LIN {X 0,Y 470.196,Z 271.556,A -85,B 0,C 180,E1 -7475.307,E2 -7475.307} C_VEL
LIN {X 0,Y 469.91,Z 283.904,A -85,B 0,C 180,E1 -7475.848,E2 -7475.848} C_VEL
LIN {X 0,Y 469.494,Z 295.789,A -85,B 0,C 180,E1 -7476.554,E2 -7476.554} C_VEL
LIN {X 0,Y 469.053,Z 307.196,A -85,B 0,C 180,E1 -7477.425,E2 -7477.425} C_VEL
LIN {X 0,Y 468.572,Z 317.556,A -85,B 0,C 180,E1 -7478.415,E2 -7478.415} C_VEL
LIN {X 0,Y 468.062,Z 326.78,A -85,B 0,C 180,E1 -7479.507,E2 -7479.507} C_VEL
LIN {X 0,Y 467.676,Z 335.773,A -85,B 0,C 180,E1 -7480.827,E2 -7480.827} C_VEL
LIN {X 0,Y 467.329,Z 343.109,A -85,B 0,C 180,E1 -7482.174,E2 -7482.174} C_VEL
LIN {X 0,Y 467.061,Z 348.773,A -85,B 0,C 180,E1 -7483.488,E2 -7483.488} C_VEL
LIN {X 0,Y 466.917,Z 353.288,A -85,B 0,C 180,E1 -7484.826,E2 -7484.826} C_VEL
LIN {X 0,Y 466.808,Z 355.68,A -85,B 0,C 180,E1 -7485.724,E2 -7485.724} C_VEL
LIN {X 0,Y 466.714,Z 357.623,A -85,B 0,C 180,E1 -7486.625,E2 -7486.625} C_VEL
LIN {X 0,Y 466.631,Z 359.065,A -85,B 0,C 180,E1 -7487.531,E2 -7487.531} C_VEL
LIN {X 0,Y 466.627,Z 360.079,A -85,B 0,C 180,E1 -7488.439,E2 -7488.439} C_VEL
LIN {X 0,Y 466.597,Z 360.681,A -85,B 0,C 180,E1 -7489.352,E2 -7489.352} C_VEL
LIN {X 0,Y 466.598,Z 360.615,A -85,B 0,C 180,E1 -7490.956,E2 -7490.956} C_VEL
LIN {X 0,Y 466.631,Z 359.745,A -85,B 0,C 180,E1 -7492.119,E2 -7492.119} C_VEL
LIN {X 0,Y 466.738,Z 358.096,A -85,B 0,C 180,E1 -7493.29,E2 -7493.29} C_VEL
LIN {X 0,Y 466.878,Z 354.549,A -85,B 0,C 180,E1 -7494.929,E2 -7494.929} C_VEL
LIN {X 0,Y 467.08,Z 350.108,A -85,B 0,C 180,E1 -7496.352,E2 -7496.352} C_VEL
LIN {X 0,Y 467.309,Z 344.226,A -85,B 0,C 180,E1 -7497.789,E2 -7497.789} C_VEL
LIN {X 0,Y 467.671,Z 337.664,A -85,B 0,C 180,E1 -7499.06,E2 -7499.06} C_VEL
LIN {X 0,Y 468.03,Z 330.441,A -85,B 0,C 180,E1 -7500.202,E2 -7500.202} C_VEL
LIN {X 0,Y 468.494,Z 321.406,A -85,B 0,C 180,E1 -7501.37,E2 -7501.37} C_VEL
LIN {X 0,Y 468.951,Z 311.594,A -85,B 0,C 180,E1 -7502.397,E2 -7502.397} C_VEL
LIN {X 0,Y 469.534,Z 300.538,A -85,B 0,C 180,E1 -7503.325,E2 -7503.325} C_VEL
LIN {X 0,Y 470.053,Z 288.74,A -85,B 0,C 180,E1 -7504.103,E2 -7504.103} C_VEL
LIN {X 0,Y 470.403,Z 275.786,A -85,B 0,C 180,E1 -7504.743,E2 -7504.743} C_VEL
LIN {X 0,Y 470.731,Z 262.741,A -85,B 0,C 180,E1 -7505.191,E2 -7505.191} C_VEL
LIN {X 0,Y 470.898,Z 248.767,A -85,B 0,C 180,E1 -7505.474,E2 -7505.474} C_VEL
LIN {X 0,Y 471.517,Z 164.162,A -85,B 0,C 180,E1 -7506.79,E2 -7506.79} C_VEL
LIN {X 0,Y 468.69,Z 150.58,A -85,B 0,C 180,E1 -7507.134,E2 -7507.134} C_VEL
LIN {X 0,Y 468.755,Z 141.458,A -85,B 0,C 180,E1 -7509.028,E2 -7509.028} C_VEL
LIN {X 0,Y 467.591,Z 135.242,A -85,B 0,C 180,E1 -7510.405,E2 -7510.405} C_VEL
LIN {X 0,Y 467.544,Z 135.249,A -85,B 0,C 180,E1 -7513.82,E2 -7513.82} C_VEL
LIN {X 0,Y 467.544,Z 135.248,A -85,B 0,C 180,E1 -7516.254,E2 -7516.254} C_VEL
LIN {X 0,Y 467.557,Z 135.241,A -85,B 0,C 180,E1 -7519.733,E2 -7519.733} C_VEL
LIN {X 0,Y 467.542,Z 135.246,A -85,B 0,C 180,E1 -7522.815,E2 -7522.815} C_VEL
LIN {X 0,Y 467.576,Z 135.239,A -85,B 0,C 180,E1 -7525.76,E2 -7525.76} C_VEL
LIN {X 0,Y 467.537,Z 135.249,A -85,B 0,C 180,E1 -7528.962,E2 -7528.962} C_VEL
LIN {X 0,Y 467.543,Z 135.245,A -85,B 0,C 180,E1 -7532.226,E2 -7532.226} C_VEL
LIN {X 0,Y 467.552,Z 135.245,A -85,B 0,C 180,E1 -7535.11,E2 -7535.11} C_VEL
LIN {X 0,Y 467.518,Z 135.243,A -85,B 0,C 180,E1 -7537.926,E2 -7537.926} C_VEL
LIN {X 0,Y 467.568,Z 135.237,A -85,B 0,C 180,E1 -7541.254,E2 -7541.254} C_VEL
LIN {X 0,Y 467.577,Z 135.242,A -85,B 0,C 180,E1 -7544.303,E2 -7544.303} C_VEL
LIN {X 0,Y 467.642,Z 135.233,A -85,B 0,C 180,E1 -7547.854,E2 -7547.854} C_VEL
LIN {X 0,Y 467.63,Z 135.231,A -85,B 0,C 180,E1 -7551.356,E2 -7551.356} C_VEL
LIN {X 0,Y 467.7,Z 135.223,A -85,B 0,C 180,E1 -7553.962,E2 -7553.962} C_VEL
LIN {X 0,Y 467.811,Z 135.208,A -85,B 0,C 180,E1 -7557.417,E2 -7557.417} C_VEL
LIN {X 0,Y 467.85,Z 135.209,A -85,B 0,C 180,E1 -7560,E2 -7560} C_VEL
LIN {X 0,Y 467.813,Z 135.203,A -85,B 0,C 180,E1 -7562.583,E2 -7562.583} C_VEL
LIN {X 0,Y 467.702,Z 135.224,A -85,B 0,C 180,E1 -7566.038,E2 -7566.038} C_VEL
LIN {X 0,Y 467.637,Z 135.227,A -85,B 0,C 180,E1 -7568.644,E2 -7568.644} C_VEL
LIN {X 0,Y 467.658,Z 135.224,A -85,B 0,C 180,E1 -7572.146,E2 -7572.146} C_VEL
LIN {X 0,Y 467.639,Z 135.233,A -85,B 0,C 180,E1 -7575.695,E2 -7575.695} C_VEL
LIN {X 0,Y 467.622,Z 135.237,A -85,B 0,C 180,E1 -7579.308,E2 -7579.308} C_VEL
LIN {X 0,Y 467.536,Z 135.237,A -85,B 0,C 180,E1 -7582.074,E2 -7582.074} C_VEL
LIN {X 0,Y 467.571,Z 135.243,A -85,B 0,C 180,E1 -7584.889,E2 -7584.889} C_VEL
LIN {X 0,Y 467.564,Z 135.24,A -85,B 0,C 180,E1 -7587.773,E2 -7587.773} C_VEL
LIN {X 0,Y 467.567,Z 135.243,A -85,B 0,C 180,E1 -7591.044,E2 -7591.044} C_VEL
LIN {X 0,Y 467.579,Z 135.237,A -85,B 0,C 180,E1 -7594.24,E2 -7594.24} C_VEL
LIN {X 0,Y 467.549,Z 135.242,A -85,B 0,C 180,E1 -7597.186,E2 -7597.186} C_VEL
LIN {X 0,Y 467.561,Z 135.244,A -85,B 0,C 180,E1 -7600.267,E2 -7600.267} C_VEL
LIN {X 0,Y 467.562,Z 135.246,A -85,B 0,C 180,E1 -7602.563,E2 -7602.563} C_VEL
LIN {X 0,Y 467.568,Z 135.242,A -85,B 0,C 180,E1 -7605.052,E2 -7605.052} C_VEL
LIN {X 0,Y 467.575,Z 135.245,A -85,B 0,C 180,E1 -7608.597,E2 -7608.597} C_VEL
LIN {X 0,Y 467.565,Z 135.244,A -85,B 0,C 180,E1 -7611.955,E2 -7611.955} C_VEL
LIN {X 0,Y 467.565,Z 135.238,A -85,B 0,C 180,E1 -7615.167,E2 -7615.167} C_VEL
LIN {X 0,Y 467.585,Z 135.243,A -85,B 0,C 180,E1 -7618.26,E2 -7618.26} C_VEL
LIN {X 0,Y 467.577,Z 135.242,A -85,B 0,C 180,E1 -7621.25,E2 -7621.25} C_VEL
LIN {X 0,Y 467.658,Z 135.282,A -85,B 0,C 180,E1 -7623.443,E2 -7623.443} C_VEL
LIN {X 0,Y 470.052,Z 147.842,A -85,B 0,C 180,E1 -7625.79,E2 -7625.79} C_VEL
LIN {X 0,Y 469.273,Z 165.112,A -85,B 0,C 180,E1 -7628.74,E2 -7628.74} C_VEL
LIN {X 0,Y 468.539,Z 183.705,A -85,B 0,C 180,E1 -7631.865,E2 -7631.865} C_VEL
LIN {X 0,Y 468.302,Z 189.868,A -85,B 0,C 180,E1 -7632.89,E2 -7632.89} C_VEL
LIN {X 0,Y 471.264,Z 209.86,A -85,B 0,C 180,E1 -7633.329,E2 -7633.329} C_VEL
LIN {X 0,Y 470.584,Z 299.18,A -85,B 0,C 180,E1 -7634.738,E2 -7634.738} C_VEL
LIN {X 0,Y 470.197,Z 312.223,A -85,B 0,C 180,E1 -7635.114,E2 -7635.114} C_VEL
LIN {X 0,Y 469.718,Z 324.844,A -85,B 0,C 180,E1 -7635.652,E2 -7635.652} C_VEL
LIN {X 0,Y 469.153,Z 336.885,A -85,B 0,C 180,E1 -7636.353,E2 -7636.353} C_VEL
LIN {X 0,Y 468.684,Z 347.532,A -85,B 0,C 180,E1 -7637.148,E2 -7637.148} C_VEL
LIN {X 0,Y 468.152,Z 358.788,A -85,B 0,C 180,E1 -7638.197,E2 -7638.197} C_VEL
LIN {X 0,Y 467.73,Z 367.295,A -85,B 0,C 180,E1 -7639.174,E2 -7639.174} C_VEL
LIN {X 0,Y 467.361,Z 375.155,A -85,B 0,C 180,E1 -7640.26,E2 -7640.26} C_VEL
LIN {X 0,Y 467.081,Z 382.844,A -85,B 0,C 180,E1 -7641.564,E2 -7641.564} C_VEL
LIN {X 0,Y 466.829,Z 389.953,A -85,B 0,C 180,E1 -7643.082,E2 -7643.082} C_VEL
LIN {X 0,Y 466.726,Z 394.684,A -85,B 0,C 180,E1 -7644.383,E2 -7644.383} C_VEL
LIN {X 0,Y 466.647,Z 398.301,A -85,B 0,C 180,E1 -7645.681,E2 -7645.681} C_VEL
LIN {X 0,Y 466.7,Z 400.168,A -85,B 0,C 180,E1 -7646.547,E2 -7646.547} C_VEL
LIN {X 0,Y 466.685,Z 401.568,A -85,B 0,C 180,E1 -7647.41,E2 -7647.41} C_VEL
LIN {X 0,Y 466.662,Z 402.568,A -85,B 0,C 180,E1 -7648.274,E2 -7648.274} C_VEL
LIN {X 0,Y 466.627,Z 403.178,A -85,B 0,C 180,E1 -7649.137,E2 -7649.137} C_VEL
LIN {X 0,Y 466.611,Z 403.388,A -85,B 0,C 180,E1 -7650,E2 -7650} C_VEL
LIN {X 0,Y 466.662,Z 402.552,A -85,B 0,C 180,E1 -7651.726,E2 -7651.726} C_VEL
LIN {X 0,Y 466.685,Z 401.548,A -85,B 0,C 180,E1 -7652.589,E2 -7652.589} C_VEL
LIN {X 0,Y 466.7,Z 400.131,A -85,B 0,C 180,E1 -7653.453,E2 -7653.453} C_VEL
LIN {X 0,Y 466.687,Z 397.162,A -85,B 0,C 180,E1 -7654.751,E2 -7654.751} C_VEL
LIN {X 0,Y 466.712,Z 392.03,A -85,B 0,C 180,E1 -7656.349,E2 -7656.349} C_VEL
LIN {X 0,Y 466.931,Z 385.925,A -85,B 0,C 180,E1 -7657.785,E2 -7657.785} C_VEL
LIN {X 0,Y 467.169,Z 378.933,A -85,B 0,C 180,E1 -7659.088,E2 -7659.088} C_VEL
LIN {X 0,Y 467.522,Z 370.162,A -85,B 0,C 180,E1 -7660.392,E2 -7660.392} C_VEL
LIN {X 0,Y 467.984,Z 361.182,A -85,B 0,C 180,E1 -7661.477,E2 -7661.477} C_VEL
LIN {X 0,Y 468.438,Z 350.306,A -85,B 0,C 180,E1 -7662.546,E2 -7662.546} C_VEL
LIN {X 0,Y 468.963,Z 338.844,A -85,B 0,C 180,E1 -7663.432,E2 -7663.432} C_VEL
LIN {X 0,Y 469.526,Z 326.234,A -85,B 0,C 180,E1 -7664.188,E2 -7664.188} C_VEL
LIN {X 0,Y 469.867,Z 315.464,A -85,B 0,C 180,E1 -7664.675,E2 -7664.675} C_VEL
LIN {X 0,Y 470.257,Z 302.801,A -85,B 0,C 180,E1 -7665.078,E2 -7665.078} C_VEL
LIN {X 0,Y 470.533,Z 286.718,A -85,B 0,C 180,E1 -7665.374,E2 -7665.374} C_VEL
LIN {X 0,Y 470.903,Z 208.82,A -85,B 0,C 180,E1 -7666.579,E2 -7666.579} C_VEL
LIN {X 0,Y 468.236,Z 190.139,A -85,B 0,C 180,E1 -7666.987,E2 -7666.987} C_VEL
LIN {X 0,Y 468.855,Z 172.415,A -85,B 0,C 180,E1 -7669.939,E2 -7669.939} C_VEL
LIN {X 0,Y 469.666,Z 153.43,A -85,B 0,C 180,E1 -7673.129,E2 -7673.129} C_VEL
LIN {X 0,Y 469.904,Z 147.289,A -85,B 0,C 180,E1 -7674.17,E2 -7674.17} C_VEL
LIN {X 0,Y 467.654,Z 135.235,A -85,B 0,C 180,E1 -7676.377,E2 -7676.377} C_VEL
LIN {X 0,Y 467.57,Z 135.242,A -85,B 0,C 180,E1 -7679.332,E2 -7679.332} C_VEL
LIN {X 0,Y 467.583,Z 135.237,A -85,B 0,C 180,E1 -7682.679,E2 -7682.679} C_VEL
LIN {X 0,Y 467.561,Z 135.245,A -85,B 0,C 180,E1 -7685.739,E2 -7685.739} C_VEL
LIN {X 0,Y 467.583,Z 135.237,A -85,B 0,C 180,E1 -7689.144,E2 -7689.144} C_VEL
LIN {X 0,Y 467.588,Z 135.236,A -85,B 0,C 180,E1 -7692.567,E2 -7692.567} C_VEL
LIN {X 0,Y 467.567,Z 135.239,A -85,B 0,C 180,E1 -7695.052,E2 -7695.052} C_VEL
LIN {X 0,Y 467.59,Z 135.241,A -85,B 0,C 180,E1 -7697.44,E2 -7697.44} C_VEL
LIN {X 0,Y 467.561,Z 135.24,A -85,B 0,C 180,E1 -7700.853,E2 -7700.853} C_VEL
LIN {X 0,Y 467.559,Z 135.24,A -85,B 0,C 180,E1 -7704.261,E2 -7704.261} C_VEL
LIN {X 0,Y 467.58,Z 135.243,A -85,B 0,C 180,E1 -7707.321,E2 -7707.321} C_VEL
LIN {X 0,Y 467.569,Z 135.239,A -85,B 0,C 180,E1 -7710.667,E2 -7710.667} C_VEL
LIN {X 0,Y 467.616,Z 135.239,A -85,B 0,C 180,E1 -7713.199,E2 -7713.199} C_VEL
LIN {X 0,Y 467.593,Z 135.236,A -85,B 0,C 180,E1 -7716.468,E2 -7716.468} C_VEL
LIN {X 0,Y 467.623,Z 135.232,A -85,B 0,C 180,E1 -7719.777,E2 -7719.777} C_VEL
LIN {X 0,Y 467.598,Z 135.236,A -85,B 0,C 180,E1 -7722.506,E2 -7722.506} C_VEL
LIN {X 0,Y 467.607,Z 135.239,A -85,B 0,C 180,E1 -7725.196,E2 -7725.196} C_VEL
LIN {X 0,Y 467.656,Z 135.227,A -85,B 0,C 180,E1 -7727.854,E2 -7727.854} C_VEL
LIN {X 0,Y 467.669,Z 135.228,A -85,B 0,C 180,E1 -7731.357,E2 -7731.357} C_VEL
LIN {X 0,Y 467.724,Z 135.219,A -85,B 0,C 180,E1 -7733.962,E2 -7733.962} C_VEL
LIN {X 0,Y 467.859,Z 135.203,A -85,B 0,C 180,E1 -7737.417,E2 -7737.417} C_VEL
LIN {X 0,Y 467.882,Z 135.2,A -85,B 0,C 180,E1 -7740,E2 -7740} C_VEL
LIN {X 0,Y 467.859,Z 135.21,A -85,B 0,C 180,E1 -7742.583,E2 -7742.583} C_VEL
LIN {X 0,Y 467.735,Z 135.219,A -85,B 0,C 180,E1 -7746.037,E2 -7746.037} C_VEL
LIN {X 0,Y 467.68,Z 135.23,A -85,B 0,C 180,E1 -7748.643,E2 -7748.643} C_VEL
LIN {X 0,Y 467.656,Z 135.232,A -85,B 0,C 180,E1 -7752.145,E2 -7752.145} C_VEL
LIN {X 0,Y 467.638,Z 135.23,A -85,B 0,C 180,E1 -7755.695,E2 -7755.695} C_VEL
LIN {X 0,Y 467.621,Z 135.231,A -85,B 0,C 180,E1 -7759.308,E2 -7759.308} C_VEL
LIN {X 0,Y 467.534,Z 135.249,A -85,B 0,C 180,E1 -7762.074,E2 -7762.074} C_VEL
LIN {X 0,Y 467.585,Z 135.236,A -85,B 0,C 180,E1 -7764.888,E2 -7764.888} C_VEL
LIN {X 0,Y 467.618,Z 135.236,A -85,B 0,C 180,E1 -7767.769,E2 -7767.769} C_VEL
LIN {X 0,Y 467.567,Z 135.238,A -85,B 0,C 180,E1 -7771.045,E2 -7771.045} C_VEL
LIN {X 0,Y 467.587,Z 135.239,A -85,B 0,C 180,E1 -7774.242,E2 -7774.242} C_VEL
LIN {X 0,Y 467.547,Z 135.242,A -85,B 0,C 180,E1 -7777.186,E2 -7777.186} C_VEL
LIN {X 0,Y 467.576,Z 135.239,A -85,B 0,C 180,E1 -7780.265,E2 -7780.265} C_VEL
LIN {X 0,Y 467.585,Z 135.236,A -85,B 0,C 180,E1 -7782.567,E2 -7782.567} C_VEL
LIN {X 0,Y 467.565,Z 135.24,A -85,B 0,C 180,E1 -7785.053,E2 -7785.053} C_VEL
LIN {X 0,Y 467.588,Z 135.242,A -85,B 0,C 180,E1 -7787.44,E2 -7787.44} C_VEL
LIN {X 0,Y 467.559,Z 135.24,A -85,B 0,C 180,E1 -7790.853,E2 -7790.853} C_VEL
LIN {X 0,Y 467.558,Z 135.24,A -85,B 0,C 180,E1 -7794.261,E2 -7794.261} C_VEL
LIN {X 0,Y 467.578,Z 135.244,A -85,B 0,C 180,E1 -7797.322,E2 -7797.322} C_VEL
LIN {X 0,Y 467.568,Z 135.239,A -85,B 0,C 180,E1 -7800.668,E2 -7800.668} C_VEL
LIN {X 0,Y 467.615,Z 135.24,A -85,B 0,C 180,E1 -7803.2,E2 -7803.2} C_VEL
LIN {X 0,Y 467.592,Z 135.236,A -85,B 0,C 180,E1 -7806.468,E2 -7806.468} C_VEL
LIN {X 0,Y 467.622,Z 135.232,A -85,B 0,C 180,E1 -7809.777,E2 -7809.777} C_VEL
LIN {X 0,Y 467.598,Z 135.236,A -85,B 0,C 180,E1 -7812.507,E2 -7812.507} C_VEL
LIN {X 0,Y 467.605,Z 135.239,A -85,B 0,C 180,E1 -7815.197,E2 -7815.197} C_VEL
LIN {X 0,Y 467.596,Z 135.237,A -85,B 0,C 180,E1 -7815.422,E2 -7815.422} C_VEL
LIN {X 0,Y 466.925,Z 135.319,A -85,B 0,C 180,E1 -7816.141,E2 -7816.141} C_VEL
LIN {X 0,Y 464.082,Z 135.676,A -85,B 0,C 180,E1 -7817.309,E2 -7817.309} C_VEL
LIN {X 0,Y 461.683,Z 135.973,A -85,B 0,C 180,E1 -7818.252,E2 -7818.252} C_VEL
LIN {X 0,Y 460.656,Z 136.106,A -85,B 0,C 180,E1 -7818.979,E2 -7818.979} C_VEL
LIN {X 0,Y 460.574,Z 136.11,A -85,B 0,C 180,E1 -7819.226,E2 -7819.226} C_VEL
LIN {X 0,Y 460.669,Z 136.103,A -85,B 0,C 180,E1 -7822.587,E2 -7822.587} C_VEL
LIN {X 0,Y 460.691,Z 136.103,A -85,B 0,C 180,E1 -7824.748,E2 -7824.748} C_VEL
LIN {X 0,Y 460.8,Z 136.086,A -85,B 0,C 180,E1 -7827.378,E2 -7827.378} C_VEL
LIN {X 0,Y 460.832,Z 136.088,A -85,B 0,C 180,E1 -7829.782,E2 -7829.782} C_VEL
LIN {X 0,Y 461.668,Z 143.128,A -85,B 0,C 180,E1 -7831.309,E2 -7831.309} C_VEL
LIN {X 0,Y 461.465,Z 150.576,A -85,B 0,C 180,E1 -7832.865,E2 -7832.865} C_VEL
LIN {X 0,Y 464.479,Z 166.22,A -85,B 0,C 180,E1 -7833.232,E2 -7833.232} C_VEL
LIN {X 0,Y 463.61,Z 257.402,A -85,B 0,C 180,E1 -7834.674,E2 -7834.674} C_VEL
LIN {X 0,Y 463.342,Z 270.667,A -85,B 0,C 180,E1 -7835.058,E2 -7835.058} C_VEL
LIN {X 0,Y 463.017,Z 283.365,A -85,B 0,C 180,E1 -7835.608,E2 -7835.608} C_VEL
LIN {X 0,Y 462.596,Z 295.48,A -85,B 0,C 180,E1 -7836.324,E2 -7836.324} C_VEL
LIN {X 0,Y 462.151,Z 306.991,A -85,B 0,C 180,E1 -7837.207,E2 -7837.207} C_VEL
LIN {X 0,Y 461.621,Z 316.821,A -85,B 0,C 180,E1 -7838.144,E2 -7838.144} C_VEL
LIN {X 0,Y 461.147,Z 325.936,A -85,B 0,C 180,E1 -7839.208,E2 -7839.208} C_VEL
LIN {X 0,Y 460.665,Z 335.146,A -85,B 0,C 180,E1 -7840.549,E2 -7840.549} C_VEL
LIN {X 0,Y 460.321,Z 342.28,A -85,B 0,C 180,E1 -7841.839,E2 -7841.839} C_VEL
LIN {X 0,Y 460.047,Z 348.506,A -85,B 0,C 180,E1 -7843.247,E2 -7843.247} C_VEL
LIN {X 0,Y 459.876,Z 353.163,A -85,B 0,C 180,E1 -7844.605,E2 -7844.605} C_VEL
LIN {X 0,Y 459.702,Z 356.698,A -85,B 0,C 180,E1 -7845.973,E2 -7845.973} C_VEL
LIN {X 0,Y 459.603,Z 358.447,A -85,B 0,C 180,E1 -7846.89,E2 -7846.89} C_VEL
LIN {X 0,Y 459.543,Z 360.487,A -85,B 0,C 180,E1 -7848.524,E2 -7848.524} C_VEL
LIN {X 0,Y 459.514,Z 361.075,A -85,B 0,C 180,E1 -7849.663,E2 -7849.663} C_VEL
LIN {X 0,Y 459.508,Z 360.881,A -85,B 0,C 180,E1 -7851.098,E2 -7851.098} C_VEL
LIN {X 0,Y 459.558,Z 359.697,A -85,B 0,C 180,E1 -7852.478,E2 -7852.478} C_VEL
LIN {X 0,Y 459.671,Z 358.257,A -85,B 0,C 180,E1 -7853.458,E2 -7853.458} C_VEL
LIN {X 0,Y 459.815,Z 355.292,A -85,B 0,C 180,E1 -7854.855,E2 -7854.855} C_VEL
LIN {X 0,Y 459.998,Z 351.028,A -85,B 0,C 180,E1 -7856.3,E2 -7856.3} C_VEL
LIN {X 0,Y 460.273,Z 344.609,A -85,B 0,C 180,E1 -7857.913,E2 -7857.913} C_VEL
LIN {X 0,Y 460.675,Z 337.949,A -85,B 0,C 180,E1 -7859.222,E2 -7859.222} C_VEL
LIN {X 0,Y 461.098,Z 330.249,A -85,B 0,C 180,E1 -7860.451,E2 -7860.451} C_VEL
LIN {X 0,Y 461.571,Z 321.633,A -85,B 0,C 180,E1 -7861.57,E2 -7861.57} C_VEL
LIN {X 0,Y 462.068,Z 311.08,A -85,B 0,C 180,E1 -7862.68,E2 -7862.68} C_VEL
LIN {X 0,Y 462.68,Z 300.588,A -85,B 0,C 180,E1 -7863.563,E2 -7863.563} C_VEL
LIN {X 0,Y 463.214,Z 288.767,A -85,B 0,C 180,E1 -7864.348,E2 -7864.348} C_VEL
LIN {X 0,Y 463.58,Z 275.971,A -85,B 0,C 180,E1 -7864.986,E2 -7864.986} C_VEL
LIN {X 0,Y 463.925,Z 262.705,A -85,B 0,C 180,E1 -7865.445,E2 -7865.445} C_VEL
LIN {X 0,Y 464.126,Z 247.598,A -85,B 0,C 180,E1 -7865.744,E2 -7865.744} C_VEL
LIN {X 0,Y 464.845,Z 165.396,A -85,B 0,C 180,E1 -7867.043,E2 -7867.043} C_VEL
LIN {X 0,Y 461.776,Z 150.914,A -85,B 0,C 180,E1 -7867.423,E2 -7867.423} C_VEL
LIN {X 0,Y 461.848,Z 142.925,A -85,B 0,C 180,E1 -7869.098,E2 -7869.098} C_VEL
LIN {X 0,Y 460.523,Z 136.122,A -85,B 0,C 180,E1 -7870.62,E2 -7870.62} C_VEL
LIN {X 0,Y 460.504,Z 136.124,A -85,B 0,C 180,E1 -7874.169,E2 -7874.169} C_VEL
LIN {X 0,Y 460.462,Z 136.131,A -85,B 0,C 180,E1 -7877.107,E2 -7877.107} C_VEL
LIN {X 0,Y 460.513,Z 136.117,A -85,B 0,C 180,E1 -7880.136,E2 -7880.136} C_VEL
LIN {X 0,Y 460.472,Z 136.122,A -85,B 0,C 180,E1 -7883.47,E2 -7883.47} C_VEL
LIN {X 0,Y 460.516,Z 136.122,A -85,B 0,C 180,E1 -7886.674,E2 -7886.674} C_VEL
LIN {X 0,Y 460.493,Z 136.123,A -85,B 0,C 180,E1 -7889.759,E2 -7889.759} C_VEL
LIN {X 0,Y 460.489,Z 136.13,A -85,B 0,C 180,E1 -7892.751,E2 -7892.751} C_VEL
LIN {X 0,Y 460.512,Z 136.12,A -85,B 0,C 180,E1 -7895.666,E2 -7895.666} C_VEL
LIN {X 0,Y 460.51,Z 136.124,A -85,B 0,C 180,E1 -7898.583,E2 -7898.583} C_VEL
LIN {X 0,Y 460.526,Z 136.114,A -85,B 0,C 180,E1 -7901.308,E2 -7901.308} C_VEL
LIN {X 0,Y 460.521,Z 136.121,A -85,B 0,C 180,E1 -7904.056,E2 -7904.056} C_VEL
LIN {X 0,Y 460.602,Z 136.108,A -85,B 0,C 180,E1 -7907.666,E2 -7907.666} C_VEL
LIN {X 0,Y 460.585,Z 136.109,A -85,B 0,C 180,E1 -7911.223,E2 -7911.223} C_VEL
LIN {X 0,Y 460.667,Z 136.098,A -85,B 0,C 180,E1 -7913.87,E2 -7913.87} C_VEL
LIN {X 0,Y 460.755,Z 136.087,A -85,B 0,C 180,E1 -7917.377,E2 -7917.377} C_VEL
LIN {X 0,Y 460.819,Z 136.085,A -85,B 0,C 180,E1 -7920,E2 -7920} C_VEL
LIN {X 0,Y 460.756,Z 136.081,A -85,B 0,C 180,E1 -7922.623,E2 -7922.623} C_VEL
LIN {X 0,Y 460.668,Z 136.099,A -85,B 0,C 180,E1 -7926.131,E2 -7926.131} C_VEL
LIN {X 0,Y 460.595,Z 136.104,A -85,B 0,C 180,E1 -7928.777,E2 -7928.777} C_VEL
LIN {X 0,Y 460.612,Z 136.101,A -85,B 0,C 180,E1 -7932.334,E2 -7932.334} C_VEL
LIN {X 0,Y 460.581,Z 136.109,A -85,B 0,C 180,E1 -7935.988,E2 -7935.988} C_VEL
LIN {X 0,Y 460.568,Z 136.114,A -85,B 0,C 180,E1 -7939.616,E2 -7939.616} C_VEL
LIN {X 0,Y 460.512,Z 136.113,A -85,B 0,C 180,E1 -7942.429,E2 -7942.429} C_VEL
LIN {X 0,Y 460.549,Z 136.111,A -85,B 0,C 180,E1 -7945.797,E2 -7945.797} C_VEL
LIN {X 0,Y 460.517,Z 136.117,A -85,B 0,C 180,E1 -7948.236,E2 -7948.236} C_VEL
LIN {X 0,Y 460.522,Z 136.12,A -85,B 0,C 180,E1 -7951.283,E2 -7951.283} C_VEL
LIN {X 0,Y 460.525,Z 136.118,A -85,B 0,C 180,E1 -7954.504,E2 -7954.504} C_VEL
LIN {X 0,Y 460.503,Z 136.118,A -85,B 0,C 180,E1 -7957.623,E2 -7957.623} C_VEL
LIN {X 0,Y 460.527,Z 136.12,A -85,B 0,C 180,E1 -7960.267,E2 -7960.267} C_VEL
LIN {X 0,Y 460.51,Z 136.119,A -85,B 0,C 180,E1 -7963.374,E2 -7963.374} C_VEL
LIN {X 0,Y 460.511,Z 136.126,A -85,B 0,C 180,E1 -7966.626,E2 -7966.626} C_VEL
LIN {X 0,Y 460.537,Z 136.119,A -85,B 0,C 180,E1 -7969.732,E2 -7969.732} C_VEL
LIN {X 0,Y 460.499,Z 136.121,A -85,B 0,C 180,E1 -7972.524,E2 -7972.524} C_VEL
LIN {X 0,Y 460.548,Z 136.114,A -85,B 0,C 180,E1 -7975.624,E2 -7975.624} C_VEL
LIN {X 0,Y 460.54,Z 136.119,A -85,B 0,C 180,E1 -7978.745,E2 -7978.745} C_VEL
LIN {X 0,Y 460.583,Z 136.115,A -85,B 0,C 180,E1 -7982.254,E2 -7982.254} C_VEL
LIN {X 0,Y 460.59,Z 136.157,A -85,B 0,C 180,E1 -7983.187,E2 -7983.187} C_VEL
LIN {X 0,Y 463.079,Z 148.727,A -85,B 0,C 180,E1 -7985.589,E2 -7985.589} C_VEL
LIN {X 0,Y 462.484,Z 162.398,A -85,B 0,C 180,E1 -7987.968,E2 -7987.968} C_VEL
LIN {X 0,Y 461.635,Z 182.163,A -85,B 0,C 180,E1 -7991.355,E2 -7991.355} C_VEL
LIN {X 0,Y 461.33,Z 189.52,A -85,B 0,C 180,E1 -7992.603,E2 -7992.603} C_VEL
LIN {X 0,Y 464.487,Z 210.587,A -85,B 0,C 180,E1 -7993.078,E2 -7993.078} C_VEL
LIN {X 0,Y 463.803,Z 298.364,A -85,B 0,C 180,E1 -7994.482,E2 -7994.482} C_VEL
LIN {X 0,Y 463.352,Z 311.564,A -85,B 0,C 180,E1 -7994.86,E2 -7994.86} C_VEL
LIN {X 0,Y 462.836,Z 324.826,A -85,B 0,C 180,E1 -7995.434,E2 -7995.434} C_VEL
LIN {X 0,Y 462.238,Z 336.776,A -85,B 0,C 180,E1 -7996.145,E2 -7996.145} C_VEL
LIN {X 0,Y 461.758,Z 347.116,A -85,B 0,C 180,E1 -7996.929,E2 -7996.929} C_VEL
LIN {X 0,Y 461.225,Z 357.534,A -85,B 0,C 180,E1 -7997.906,E2 -7997.906} C_VEL
LIN {X 0,Y 460.743,Z 367.089,A -85,B 0,C 180,E1 -7999.008,E2 -7999.008} C_VEL
LIN {X 0,Y 460.262,Z 376.295,A -85,B 0,C 180,E1 -8000.33,E2 -8000.33} C_VEL
LIN {X 0,Y 459.964,Z 383.721,A -85,B 0,C 180,E1 -8001.654,E2 -8001.654} C_VEL
LIN {X 0,Y 459.741,Z 389.689,A -85,B 0,C 180,E1 -8002.975,E2 -8002.975} C_VEL
LIN {X 0,Y 459.625,Z 394.408,A -85,B 0,C 180,E1 -8004.296,E2 -8004.296} C_VEL
LIN {X 0,Y 459.565,Z 398.013,A -85,B 0,C 180,E1 -8005.615,E2 -8005.615} C_VEL
LIN {X 0,Y 459.596,Z 399.87,A -85,B 0,C 180,E1 -8006.493,E2 -8006.493} C_VEL
LIN {X 0,Y 459.605,Z 401.263,A -85,B 0,C 180,E1 -8007.371,E2 -8007.371} C_VEL
LIN {X 0,Y 459.56,Z 402.863,A -85,B 0,C 180,E1 -8009.124,E2 -8009.124} C_VEL
LIN {X 0,Y 459.542,Z 403.063,A -85,B 0,C 180,E1 -8010,E2 -8010} C_VEL
LIN {X 0,Y 459.56,Z 402.833,A -85,B 0,C 180,E1 -8010.876,E2 -8010.876} C_VEL
LIN {X 0,Y 459.605,Z 401.204,A -85,B 0,C 180,E1 -8012.629,E2 -8012.629} C_VEL
LIN {X 0,Y 459.597,Z 399.774,A -85,B 0,C 180,E1 -8013.507,E2 -8013.507} C_VEL
LIN {X 0,Y 459.614,Z 396.793,A -85,B 0,C 180,E1 -8014.824,E2 -8014.824} C_VEL
LIN {X 0,Y 459.635,Z 392.029,A -85,B 0,C 180,E1 -8016.342,E2 -8016.342} C_VEL
LIN {X 0,Y 459.867,Z 385.519,A -85,B 0,C 180,E1 -8017.906,E2 -8017.906} C_VEL
LIN {X 0,Y 460.104,Z 378.501,A -85,B 0,C 180,E1 -8019.229,E2 -8019.229} C_VEL
LIN {X 0,Y 460.496,Z 369.702,A -85,B 0,C 180,E1 -8020.553,E2 -8020.553} C_VEL
LIN {X 0,Y 461.057,Z 359.711,A -85,B 0,C 180,E1 -8021.764,E2 -8021.764} C_VEL
LIN {X 0,Y 461.461,Z 349.611,A -85,B 0,C 180,E1 -8022.752,E2 -8022.752} C_VEL
LIN {X 0,Y 462.017,Z 338.251,A -85,B 0,C 180,E1 -8023.637,E2 -8023.637} C_VEL
LIN {X 0,Y 462.585,Z 325.566,A -85,B 0,C 180,E1 -8024.405,E2 -8024.405} C_VEL
LIN {X 0,Y 463.059,Z 313.187,A -85,B 0,C 180,E1 -8024.952,E2 -8024.952} C_VEL
LIN {X 0,Y 463.496,Z 300.581,A -85,B 0,C 180,E1 -8025.331,E2 -8025.331} C_VEL
LIN {X 0,Y 463.717,Z 279.848,A -85,B 0,C 180,E1 -8025.69,E2 -8025.69} C_VEL
LIN {X 0,Y 464.044,Z 209.571,A -85,B 0,C 180,E1 -8026.796,E2 -8026.796} C_VEL
LIN {X 0,Y 461.224,Z 189.903,A -85,B 0,C 180,E1 -8027.224,E2 -8027.224} C_VEL
LIN {X 0,Y 461.85,Z 171.964,A -85,B 0,C 180,E1 -8030.254,E2 -8030.254} C_VEL
LIN {X 0,Y 462.717,Z 154.319,A -85,B 0,C 180,E1 -8033.26,E2 -8033.26} C_VEL
LIN {X 0,Y 462.864,Z 148.003,A -85,B 0,C 180,E1 -8034.352,E2 -8034.352} C_VEL
LIN {X 0,Y 460.616,Z 136.111,A -85,B 0,C 180,E1 -8036.567,E2 -8036.567} C_VEL
LIN {X 0,Y 460.532,Z 136.12,A -85,B 0,C 180,E1 -8039.558,E2 -8039.558} C_VEL
LIN {X 0,Y 460.533,Z 136.119,A -85,B 0,C 180,E1 -8042.284,E2 -8042.284} C_VEL
LIN {X 0,Y 460.511,Z 136.119,A -85,B 0,C 180,E1 -8045.445,E2 -8045.445} C_VEL
LIN {X 0,Y 460.546,Z 136.113,A -85,B 0,C 180,E1 -8048.897,E2 -8048.897} C_VEL
LIN {X 0,Y 460.524,Z 136.119,A -85,B 0,C 180,E1 -8052.181,E2 -8052.181} C_VEL
LIN {X 0,Y 460.515,Z 136.121,A -85,B 0,C 180,E1 -8055.411,E2 -8055.411} C_VEL
LIN {X 0,Y 460.533,Z 136.115,A -85,B 0,C 180,E1 -8058.397,E2 -8058.397} C_VEL
LIN {X 0,Y 460.519,Z 136.12,A -85,B 0,C 180,E1 -8061.266,E2 -8061.266} C_VEL
LIN {X 0,Y 460.509,Z 136.118,A -85,B 0,C 180,E1 -8064.554,E2 -8064.554} C_VEL
LIN {X 0,Y 460.53,Z 136.119,A -85,B 0,C 180,E1 -8067.715,E2 -8067.715} C_VEL
LIN {X 0,Y 460.54,Z 136.115,A -85,B 0,C 180,E1 -8070.769,E2 -8070.769} C_VEL
LIN {X 0,Y 460.56,Z 136.114,A -85,B 0,C 180,E1 -8073.734,E2 -8073.734} C_VEL
LIN {X 0,Y 460.546,Z 136.114,A -85,B 0,C 180,E1 -8076.624,E2 -8076.624} C_VEL
LIN {X 0,Y 460.552,Z 136.116,A -85,B 0,C 180,E1 -8079.453,E2 -8079.453} C_VEL
LIN {X 0,Y 460.549,Z 136.113,A -85,B 0,C 180,E1 -8082.23,E2 -8082.23} C_VEL
LIN {X 0,Y 460.566,Z 136.118,A -85,B 0,C 180,E1 -8084.965,E2 -8084.965} C_VEL
LIN {X 0,Y 460.61,Z 136.108,A -85,B 0,C 180,E1 -8088.559,E2 -8088.559} C_VEL
LIN {X 0,Y 460.619,Z 136.107,A -85,B 0,C 180,E1 -8091.224,E2 -8091.224} C_VEL
LIN {X 0,Y 460.688,Z 136.095,A -85,B 0,C 180,E1 -8093.87,E2 -8093.87} C_VEL
LIN {X 0,Y 460.8,Z 136.082,A -85,B 0,C 180,E1 -8097.377,E2 -8097.377} C_VEL
LIN {X 0,Y 460.853,Z 136.075,A -85,B 0,C 180,E1 -8100,E2 -8100} C_VEL
LIN {X 0,Y 460.824,Z 136.087,A -85,B 0,C 180,E1 -8102.622,E2 -8102.622} C_VEL
LIN {X 0,Y 460.701,Z 136.096,A -85,B 0,C 180,E1 -8106.13,E2 -8106.13} C_VEL
LIN {X 0,Y 460.627,Z 136.107,A -85,B 0,C 180,E1 -8108.776,E2 -8108.776} C_VEL
LIN {X 0,Y 460.613,Z 136.112,A -85,B 0,C 180,E1 -8112.445,E2 -8112.445} C_VEL
LIN {X 0,Y 460.6,Z 136.11,A -85,B 0,C 180,E1 -8115.997,E2 -8115.997} C_VEL
LIN {X 0,Y 460.567,Z 136.111,A -85,B 0,C 180,E1 -8119.615,E2 -8119.615} C_VEL
LIN {X 0,Y 460.51,Z 136.122,A -85,B 0,C 180,E1 -8122.429,E2 -8122.429} C_VEL
LIN {X 0,Y 460.552,Z 136.116,A -85,B 0,C 180,E1 -8125.798,E2 -8125.798} C_VEL
LIN {X 0,Y 460.55,Z 136.118,A -85,B 0,C 180,E1 -8128.233,E2 -8128.233} C_VEL
LIN {X 0,Y 460.519,Z 136.117,A -85,B 0,C 180,E1 -8131.283,E2 -8131.283} C_VEL
LIN {X 0,Y 460.53,Z 136.116,A -85,B 0,C 180,E1 -8134.505,E2 -8134.505} C_VEL
LIN {X 0,Y 460.5,Z 136.124,A -85,B 0,C 180,E1 -8137.623,E2 -8137.623} C_VEL
LIN {X 0,Y 460.541,Z 136.116,A -85,B 0,C 180,E1 -8140.269,E2 -8140.269} C_VEL
LIN {X 0,Y 460.497,Z 136.123,A -85,B 0,C 180,E1 -8143.376,E2 -8143.376} C_VEL
LIN {X 0,Y 460.497,Z 136.119,A -85,B 0,C 180,E1 -8146.625,E2 -8146.625} C_VEL
LIN {X 0,Y 460.538,Z 136.12,A -85,B 0,C 180,E1 -8149.731,E2 -8149.731} C_VEL
LIN {X 0,Y 460.498,Z 136.119,A -85,B 0,C 180,E1 -8152.524,E2 -8152.524} C_VEL
LIN {X 0,Y 460.536,Z 136.119,A -85,B 0,C 180,E1 -8155.623,E2 -8155.623} C_VEL
LIN {X 0,Y 460.536,Z 136.115,A -85,B 0,C 180,E1 -8158.745,E2 -8158.745} C_VEL
LIN {X 0,Y 460.58,Z 136.109,A -85,B 0,C 180,E1 -8162.254,E2 -8162.254} C_VEL
LIN {X 0,Y 460.546,Z 136.115,A -85,B 0,C 180,E1 -8164.705,E2 -8164.705} C_VEL
LIN {X 0,Y 460.51,Z 136.12,A -85,B 0,C 180,E1 -8167.571,E2 -8167.571} C_VEL
LIN {X 0,Y 460.568,Z 136.111,A -85,B 0,C 180,E1 -8170.385,E2 -8170.385} C_VEL
LIN {X 0,Y 460.604,Z 136.106,A -85,B 0,C 180,E1 -8174.059,E2 -8174.059} C_VEL
LIN {X 0,Y 460.609,Z 136.106,A -85,B 0,C 180,E1 -8177.666,E2 -8177.666} C_VEL
LIN {X 0,Y 460.574,Z 136.11,A -85,B 0,C 180,E1 -8179.226,E2 -8179.226} C_VEL
LIN {X 0,Y 459.911,Z 136.195,A -85,B 0,C 180,E1 -8179.955,E2 -8179.955} C_VEL
LIN {X 0,Y 457.07,Z 136.556,A -85,B 0,C 180,E1 -8181.141,E2 -8181.141} C_VEL
LIN {X 0,Y 454.679,Z 136.855,A -85,B 0,C 180,E1 -8182.098,E2 -8182.098} C_VEL
LIN {X 0,Y 453.669,Z 136.977,A -85,B 0,C 180,E1 -8182.836,E2 -8182.836} C_VEL
LIN {X 0,Y 453.596,Z 136.983,A -85,B 0,C 180,E1 -8183.087,E2 -8183.087} C_VEL
LIN {X 0,Y 453.663,Z 136.977,A -85,B 0,C 180,E1 -8184.667,E2 -8184.667} C_VEL
LIN {X 0,Y 453.744,Z 136.965,A -85,B 0,C 180,E1 -8187.337,E2 -8187.337} C_VEL
LIN {X 0,Y 453.796,Z 137.063,A -85,B 0,C 180,E1 -8189.64,E2 -8189.64} C_VEL
LIN {X 0,Y 454.688,Z 143.726,A -85,B 0,C 180,E1 -8191.107,E2 -8191.107} C_VEL
LIN {X 0,Y 454.551,Z 151.068,A -85,B 0,C 180,E1 -8192.631,E2 -8192.631} C_VEL
LIN {X 0,Y 457.642,Z 166.686,A -85,B 0,C 180,E1 -8192.997,E2 -8192.997} C_VEL
LIN {X 0,Y 456.721,Z 258.225,A -85,B 0,C 180,E1 -8194.468,E2 -8194.468} C_VEL
LIN {X 0,Y 456.451,Z 271.307,A -85,B 0,C 180,E1 -8194.858,E2 -8194.858} C_VEL
LIN {X 0,Y 456.131,Z 283.902,A -85,B 0,C 180,E1 -8195.415,E2 -8195.415} C_VEL
LIN {X 0,Y 455.706,Z 295.17,A -85,B 0,C 180,E1 -8196.087,E2 -8196.087} C_VEL
LIN {X 0,Y 455.245,Z 306.79,A -85,B 0,C 180,E1 -8196.983,E2 -8196.983} C_VEL
LIN {X 0,Y 454.636,Z 317.325,A -85,B 0,C 180,E1 -8197.997,E2 -8197.997} C_VEL
LIN {X 0,Y 454.133,Z 326.762,A -85,B 0,C 180,E1 -8199.127,E2 -8199.127} C_VEL
LIN {X 0,Y 453.623,Z 335.885,A -85,B 0,C 180,E1 -8200.489,E2 -8200.489} C_VEL
LIN {X 0,Y 453.228,Z 343.737,A -85,B 0,C 180,E1 -8201.962,E2 -8201.962} C_VEL
LIN {X 0,Y 452.943,Z 349.914,A -85,B 0,C 180,E1 -8203.459,E2 -8203.459} C_VEL
LIN {X 0,Y 452.748,Z 354.325,A -85,B 0,C 180,E1 -8204.841,E2 -8204.841} C_VEL
LIN {X 0,Y 452.587,Z 357.627,A -85,B 0,C 180,E1 -8206.231,E2 -8206.231} C_VEL
LIN {X 0,Y 452.487,Z 359.268,A -85,B 0,C 180,E1 -8207.164,E2 -8207.164} C_VEL
LIN {X 0,Y 452.448,Z 360.922,A -85,B 0,C 180,E1 -8208.643,E2 -8208.643} C_VEL
LIN {X 0,Y 452.409,Z 361.459,A -85,B 0,C 180,E1 -8209.984,E2 -8209.984} C_VEL
LIN {X 0,Y 452.427,Z 361.146,A -85,B 0,C 180,E1 -8211.245,E2 -8211.245} C_VEL
LIN {X 0,Y 452.524,Z 359.633,A -85,B 0,C 180,E1 -8212.847,E2 -8212.847} C_VEL
LIN {X 0,Y 452.685,Z 357.126,A -85,B 0,C 180,E1 -8214.294,E2 -8214.294} C_VEL
LIN {X 0,Y 452.861,Z 353.212,A -85,B 0,C 180,E1 -8215.828,E2 -8215.828} C_VEL
LIN {X 0,Y 453.112,Z 348.38,A -85,B 0,C 180,E1 -8217.23,E2 -8217.23} C_VEL
LIN {X 0,Y 453.466,Z 341.793,A -85,B 0,C 180,E1 -8218.715,E2 -8218.715} C_VEL
LIN {X 0,Y 453.903,Z 334.725,A -85,B 0,C 180,E1 -8219.987,E2 -8219.987} C_VEL
LIN {X 0,Y 454.397,Z 326.406,A -85,B 0,C 180,E1 -8221.207,E2 -8221.207} C_VEL
LIN {X 0,Y 454.938,Z 317.254,A -85,B 0,C 180,E1 -8222.298,E2 -8222.298} C_VEL
LIN {X 0,Y 455.421,Z 307.863,A -85,B 0,C 180,E1 -8223.219,E2 -8223.219} C_VEL
LIN {X 0,Y 456.04,Z 296.738,A -85,B 0,C 180,E1 -8224.096,E2 -8224.096} C_VEL
LIN {X 0,Y 456.564,Z 284.93,A -85,B 0,C 180,E1 -8224.824,E2 -8224.824} C_VEL
LIN {X 0,Y 456.922,Z 272.07,A -85,B 0,C 180,E1 -8225.407,E2 -8225.407} C_VEL
LIN {X 0,Y 457.237,Z 258.917,A -85,B 0,C 180,E1 -8225.806,E2 -8225.806} C_VEL
LIN {X 0,Y 458.095,Z 166.277,A -85,B 0,C 180,E1 -8227.321,E2 -8227.321} C_VEL
LIN {X 0,Y 454.87,Z 151.208,A -85,B 0,C 180,E1 -8227.732,E2 -8227.732} C_VEL
LIN {X 0,Y 454.988,Z 145.156,A -85,B 0,C 180,E1 -8229.01,E2 -8229.01} C_VEL
LIN {X 0,Y 453.472,Z 137,A -85,B 0,C 180,E1 -8230.844,E2 -8230.844} C_VEL
LIN {X 0,Y 453.481,Z 137,A -85,B 0,C 180,E1 -8234.529,E2 -8234.529} C_VEL
LIN {X 0,Y 453.436,Z 137.004,A -85,B 0,C 180,E1 -8238.071,E2 -8238.071} C_VEL
LIN {X 0,Y 453.447,Z 136.999,A -85,B 0,C 180,E1 -8240.801,E2 -8240.801} C_VEL
LIN {X 0,Y 453.451,Z 136.995,A -85,B 0,C 180,E1 -8243.917,E2 -8243.917} C_VEL
LIN {X 0,Y 453.472,Z 137.002,A -85,B 0,C 180,E1 -8247.15,E2 -8247.15} C_VEL
LIN {X 0,Y 453.454,Z 137.002,A -85,B 0,C 180,E1 -8250.267,E2 -8250.267} C_VEL
LIN {X 0,Y 453.426,Z 137.003,A -85,B 0,C 180,E1 -8253.289,E2 -8253.289} C_VEL
LIN {X 0,Y 453.48,Z 136.999,A -85,B 0,C 180,E1 -8256.238,E2 -8256.238} C_VEL
LIN {X 0,Y 453.437,Z 137.002,A -85,B 0,C 180,E1 -8259.116,E2 -8259.116} C_VEL
LIN {X 0,Y 453.456,Z 136.996,A -85,B 0,C 180,E1 -8261.942,E2 -8261.942} C_VEL
LIN {X 0,Y 453.485,Z 136.993,A -85,B 0,C 180,E1 -8264.725,E2 -8264.725} C_VEL
LIN {X 0,Y 453.566,Z 136.984,A -85,B 0,C 180,E1 -8267.471,E2 -8267.471} C_VEL
LIN {X 0,Y 453.555,Z 136.984,A -85,B 0,C 180,E1 -8271.086,E2 -8271.086} C_VEL
LIN {X 0,Y 453.635,Z 136.973,A -85,B 0,C 180,E1 -8273.774,E2 -8273.774} C_VEL
LIN {X 0,Y 453.701,Z 136.965,A -85,B 0,C 180,E1 -8277.337,E2 -8277.337} C_VEL
LIN {X 0,Y 453.768,Z 136.963,A -85,B 0,C 180,E1 -8280,E2 -8280} C_VEL
LIN {X 0,Y 453.703,Z 136.96,A -85,B 0,C 180,E1 -8282.664,E2 -8282.664} C_VEL
LIN {X 0,Y 453.636,Z 136.974,A -85,B 0,C 180,E1 -8286.226,E2 -8286.226} C_VEL
LIN {X 0,Y 453.567,Z 136.98,A -85,B 0,C 180,E1 -8288.914,E2 -8288.914} C_VEL
LIN {X 0,Y 453.566,Z 136.979,A -85,B 0,C 180,E1 -8292.529,E2 -8292.529} C_VEL
LIN {X 0,Y 453.539,Z 136.986,A -85,B 0,C 180,E1 -8296.196,E2 -8296.196} C_VEL
LIN {X 0,Y 453.519,Z 136.99,A -85,B 0,C 180,E1 -8299.039,E2 -8299.039} C_VEL
LIN {X 0,Y 453.479,Z 136.989,A -85,B 0,C 180,E1 -8301.836,E2 -8301.836} C_VEL
LIN {X 0,Y 453.496,Z 136.995,A -85,B 0,C 180,E1 -8304.736,E2 -8304.736} C_VEL
LIN {X 0,Y 453.478,Z 136.994,A -85,B 0,C 180,E1 -8307.946,E2 -8307.946} C_VEL
LIN {X 0,Y 453.476,Z 136.996,A -85,B 0,C 180,E1 -8310.76,E2 -8310.76} C_VEL
LIN {X 0,Y 453.47,Z 136.993,A -85,B 0,C 180,E1 -8313.914,E2 -8313.914} C_VEL
LIN {X 0,Y 453.454,Z 136.998,A -85,B 0,C 180,E1 -8317.19,E2 -8317.19} C_VEL
LIN {X 0,Y 453.472,Z 137,A -85,B 0,C 180,E1 -8320.612,E2 -8320.612} C_VEL
LIN {X 0,Y 453.462,Z 137.001,A -85,B 0,C 180,E1 -8324.222,E2 -8324.222} C_VEL
LIN {X 0,Y 453.451,Z 137.002,A -85,B 0,C 180,E1 -8327.003,E2 -8327.003} C_VEL
LIN {X 0,Y 453.496,Z 136.995,A -85,B 0,C 180,E1 -8329.409,E2 -8329.409} C_VEL
LIN {X 0,Y 453.452,Z 136.999,A -85,B 0,C 180,E1 -8332.81,E2 -8332.81} C_VEL
LIN {X 0,Y 453.479,Z 136.998,A -85,B 0,C 180,E1 -8336.087,E2 -8336.087} C_VEL
LIN {X 0,Y 453.479,Z 136.999,A -85,B 0,C 180,E1 -8339.24,E2 -8339.24} C_VEL
LIN {X 0,Y 453.539,Z 136.992,A -85,B 0,C 180,E1 -8342.298,E2 -8342.298} C_VEL
LIN {X 0,Y 453.556,Z 137.057,A -85,B 0,C 180,E1 -8342.924,E2 -8342.924} C_VEL
LIN {X 0,Y 456.109,Z 149.799,A -85,B 0,C 180,E1 -8345.416,E2 -8345.416} C_VEL
LIN {X 0,Y 455.954,Z 156.517,A -85,B 0,C 180,E1 -8346.615,E2 -8346.615} C_VEL
LIN {X 0,Y 454.958,Z 175.293,A -85,B 0,C 180,E1 -8349.897,E2 -8349.897} C_VEL
LIN {X 0,Y 454.428,Z 189.457,A -85,B 0,C 180,E1 -8352.308,E2 -8352.308} C_VEL
LIN {X 0,Y 457.789,Z 211.727,A -85,B 0,C 180,E1 -8352.821,E2 -8352.821} C_VEL
LIN {X 0,Y 457.026,Z 297.658,A -85,B 0,C 180,E1 -8354.217,E2 -8354.217} C_VEL
LIN {X 0,Y 456.544,Z 310.959,A -85,B 0,C 180,E1 -8354.6,E2 -8354.6} C_VEL
LIN {X 0,Y 456.033,Z 323.703,A -85,B 0,C 180,E1 -8355.154,E2 -8355.154} C_VEL
LIN {X 0,Y 455.467,Z 335.074,A -85,B 0,C 180,E1 -8355.821,E2 -8355.821} C_VEL
LIN {X 0,Y 454.823,Z 346.95,A -85,B 0,C 180,E1 -8356.724,E2 -8356.724} C_VEL
LIN {X 0,Y 454.257,Z 357.354,A -85,B 0,C 180,E1 -8357.717,E2 -8357.717} C_VEL
LIN {X 0,Y 453.761,Z 366.881,A -85,B 0,C 180,E1 -8358.837,E2 -8358.837} C_VEL
LIN {X 0,Y 453.222,Z 376.061,A -85,B 0,C 180,E1 -8360.179,E2 -8360.179} C_VEL
LIN {X 0,Y 452.921,Z 383.472,A -85,B 0,C 180,E1 -8361.523,E2 -8361.523} C_VEL
LIN {X 0,Y 452.669,Z 389.426,A -85,B 0,C 180,E1 -8362.865,E2 -8362.865} C_VEL
LIN {X 0,Y 452.527,Z 394.132,A -85,B 0,C 180,E1 -8364.206,E2 -8364.206} C_VEL
LIN {X 0,Y 452.486,Z 397.726,A -85,B 0,C 180,E1 -8365.546,E2 -8365.546} C_VEL
LIN {X 0,Y 452.493,Z 399.57,A -85,B 0,C 180,E1 -8366.438,E2 -8366.438} C_VEL
LIN {X 0,Y 452.527,Z 400.959,A -85,B 0,C 180,E1 -8367.329,E2 -8367.329} C_VEL
LIN {X 0,Y 452.494,Z 402.549,A -85,B 0,C 180,E1 -8369.11,E2 -8369.11} C_VEL
LIN {X 0,Y 452.475,Z 402.738,A -85,B 0,C 180,E1 -8370,E2 -8370} C_VEL
LIN {X 0,Y 452.494,Z 402.501,A -85,B 0,C 180,E1 -8370.89,E2 -8370.89} C_VEL
LIN {X 0,Y 452.527,Z 400.859,A -85,B 0,C 180,E1 -8372.67,E2 -8372.67} C_VEL
LIN {X 0,Y 452.495,Z 399.415,A -85,B 0,C 180,E1 -8373.562,E2 -8373.562} C_VEL
LIN {X 0,Y 452.541,Z 396.424,A -85,B 0,C 180,E1 -8374.9,E2 -8374.9} C_VEL
LIN {X 0,Y 452.554,Z 392.043,A -85,B 0,C 180,E1 -8376.331,E2 -8376.331} C_VEL
LIN {X 0,Y 452.757,Z 386.13,A -85,B 0,C 180,E1 -8377.806,E2 -8377.806} C_VEL
LIN {X 0,Y 453.009,Z 379.329,A -85,B 0,C 180,E1 -8379.15,E2 -8379.15} C_VEL
LIN {X 0,Y 453.404,Z 370.881,A -85,B 0,C 180,E1 -8380.494,E2 -8380.494} C_VEL
LIN {X 0,Y 453.898,Z 362.174,A -85,B 0,C 180,E1 -8381.612,E2 -8381.612} C_VEL
LIN {X 0,Y 454.368,Z 351.969,A -85,B 0,C 180,E1 -8382.683,E2 -8382.683} C_VEL
LIN {X 0,Y 454.951,Z 340.791,A -85,B 0,C 180,E1 -8383.626,E2 -8383.626} C_VEL
LIN {X 0,Y 455.517,Z 328.905,A -85,B 0,C 180,E1 -8384.406,E2 -8384.406} C_VEL
LIN {X 0,Y 455.975,Z 316.54,A -85,B 0,C 180,E1 -8385.018,E2 -8385.018} C_VEL
LIN {X 0,Y 456.468,Z 303.895,A -85,B 0,C 180,E1 -8385.459,E2 -8385.459} C_VEL
LIN {X 0,Y 456.71,Z 290.776,A -85,B 0,C 180,E1 -8385.737,E2 -8385.737} C_VEL
LIN {X 0,Y 457.261,Z 210.701,A -85,B 0,C 180,E1 -8387.011,E2 -8387.011} C_VEL
LIN {X 0,Y 454.228,Z 189.623,A -85,B 0,C 180,E1 -8387.467,E2 -8387.467} C_VEL
LIN {X 0,Y 454.849,Z 172.842,A -85,B 0,C 180,E1 -8390.344,E2 -8390.344} C_VEL
LIN {X 0,Y 455.766,Z 155.209,A -85,B 0,C 180,E1 -8393.395,E2 -8393.395} C_VEL
LIN {X 0,Y 455.808,Z 148.762,A -85,B 0,C 180,E1 -8394.534,E2 -8394.534} C_VEL
LIN {X 0,Y 453.567,Z 136.988,A -85,B 0,C 180,E1 -8396.764,E2 -8396.764} C_VEL
LIN {X 0,Y 453.473,Z 137.002,A -85,B 0,C 180,E1 -8399.784,E2 -8399.784} C_VEL
LIN {X 0,Y 453.492,Z 136.992,A -85,B 0,C 180,E1 -8403.189,E2 -8403.189} C_VEL
LIN {X 0,Y 453.454,Z 136.999,A -85,B 0,C 180,E1 -8406.299,E2 -8406.299} C_VEL
LIN {X 0,Y 453.518,Z 136.991,A -85,B 0,C 180,E1 -8409.447,E2 -8409.447} C_VEL
LIN {X 0,Y 453.463,Z 136.996,A -85,B 0,C 180,E1 -8412.995,E2 -8412.995} C_VEL
LIN {X 0,Y 453.464,Z 137.002,A -85,B 0,C 180,E1 -8415.778,E2 -8415.778} C_VEL
LIN {X 0,Y 453.48,Z 136.995,A -85,B 0,C 180,E1 -8418.209,E2 -8418.209} C_VEL
LIN {X 0,Y 453.488,Z 136.993,A -85,B 0,C 180,E1 -8420.794,E2 -8420.794} C_VEL
LIN {X 0,Y 453.454,Z 136.999,A -85,B 0,C 180,E1 -8423.917,E2 -8423.917} C_VEL
LIN {X 0,Y 453.479,Z 136.997,A -85,B 0,C 180,E1 -8427.151,E2 -8427.151} C_VEL
LIN {X 0,Y 453.475,Z 136.994,A -85,B 0,C 180,E1 -8430.268,E2 -8430.268} C_VEL
LIN {X 0,Y 453.505,Z 136.998,A -85,B 0,C 180,E1 -8433.294,E2 -8433.294} C_VEL
LIN {X 0,Y 453.502,Z 136.99,A -85,B 0,C 180,E1 -8436.239,E2 -8436.239} C_VEL
LIN {X 0,Y 453.483,Z 137,A -85,B 0,C 180,E1 -8439.117,E2 -8439.117} C_VEL
LIN {X 0,Y 453.504,Z 136.99,A -85,B 0,C 180,E1 -8441.944,E2 -8441.944} C_VEL
LIN {X 0,Y 453.54,Z 136.99,A -85,B 0,C 180,E1 -8444.726,E2 -8444.726} C_VEL
LIN {X 0,Y 453.559,Z 136.985,A -85,B 0,C 180,E1 -8448.379,E2 -8448.379} C_VEL
LIN {X 0,Y 453.585,Z 136.985,A -85,B 0,C 180,E1 -8451.086,E2 -8451.086} C_VEL
LIN {X 0,Y 453.653,Z 136.972,A -85,B 0,C 180,E1 -8453.774,E2 -8453.774} C_VEL
LIN {X 0,Y 453.744,Z 136.962,A -85,B 0,C 180,E1 -8457.337,E2 -8457.337} C_VEL
LIN {X 0,Y 453.823,Z 136.951,A -85,B 0,C 180,E1 -8460,E2 -8460} C_VEL
LIN {X 0,Y 453.764,Z 136.965,A -85,B 0,C 180,E1 -8462.663,E2 -8462.663} C_VEL
LIN {X 0,Y 453.669,Z 136.973,A -85,B 0,C 180,E1 -8466.225,E2 -8466.225} C_VEL
LIN {X 0,Y 453.59,Z 136.982,A -85,B 0,C 180,E1 -8468.913,E2 -8468.913} C_VEL
LIN {X 0,Y 453.563,Z 136.989,A -85,B 0,C 180,E1 -8472.529,E2 -8472.529} C_VEL
LIN {X 0,Y 453.544,Z 136.992,A -85,B 0,C 180,E1 -8476.196,E2 -8476.196} C_VEL
LIN {X 0,Y 453.516,Z 136.989,A -85,B 0,C 180,E1 -8479.039,E2 -8479.039} C_VEL
LIN {X 0,Y 453.476,Z 136.997,A -85,B 0,C 180,E1 -8481.836,E2 -8481.836} C_VEL
LIN {X 0,Y 453.5,Z 136.992,A -85,B 0,C 180,E1 -8484.735,E2 -8484.735} C_VEL
LIN {X 0,Y 453.53,Z 136.994,A -85,B 0,C 180,E1 -8487.959,E2 -8487.959} C_VEL
LIN {X 0,Y 453.465,Z 136.998,A -85,B 0,C 180,E1 -8491.525,E2 -8491.525} C_VEL
LIN {X 0,Y 453.486,Z 136.992,A -85,B 0,C 180,E1 -8494.777,E2 -8494.777} C_VEL
LIN {X 0,Y 453.463,Z 136.997,A -85,B 0,C 180,E1 -8498.312,E2 -8498.312} C_VEL
LIN {X 0,Y 453.493,Z 136.992,A -85,B 0,C 180,E1 -8500.609,E2 -8500.609} C_VEL
LIN {X 0,Y 453.453,Z 136.999,A -85,B 0,C 180,E1 -8503.244,E2 -8503.244} C_VEL
LIN {X 0,Y 453.462,Z 137.001,A -85,B 0,C 180,E1 -8505.779,E2 -8505.779} C_VEL
LIN {X 0,Y 453.478,Z 136.995,A -85,B 0,C 180,E1 -8508.209,E2 -8508.209} C_VEL
LIN {X 0,Y 453.486,Z 136.993,A -85,B 0,C 180,E1 -8510.795,E2 -8510.795} C_VEL
LIN {X 0,Y 453.453,Z 136.999,A -85,B 0,C 180,E1 -8513.917,E2 -8513.917} C_VEL
LIN {X 0,Y 453.478,Z 136.998,A -85,B 0,C 180,E1 -8517.151,E2 -8517.151} C_VEL
LIN {X 0,Y 453.473,Z 136.994,A -85,B 0,C 180,E1 -8520.268,E2 -8520.268} C_VEL
LIN {X 0,Y 453.504,Z 136.998,A -85,B 0,C 180,E1 -8523.294,E2 -8523.294} C_VEL
LIN {X 0,Y 453.502,Z 136.99,A -85,B 0,C 180,E1 -8526.239,E2 -8526.239} C_VEL
LIN {X 0,Y 453.483,Z 137.001,A -85,B 0,C 180,E1 -8529.118,E2 -8529.118} C_VEL
LIN {X 0,Y 453.503,Z 136.99,A -85,B 0,C 180,E1 -8531.944,E2 -8531.944} C_VEL
LIN {X 0,Y 453.539,Z 136.99,A -85,B 0,C 180,E1 -8534.726,E2 -8534.726} C_VEL
LIN {X 0,Y 453.559,Z 136.985,A -85,B 0,C 180,E1 -8538.379,E2 -8538.379} C_VEL
LIN {X 0,Y 453.585,Z 136.985,A -85,B 0,C 180,E1 -8541.087,E2 -8541.087} C_VEL
LIN {X 0,Y 453.596,Z 136.983,A -85,B 0,C 180,E1 -8543.087,E2 -8543.087} C_VEL
LIN {X 0,Y 452.927,Z 137.063,A -85,B 0,C 180,E1 -8543.827,E2 -8543.827} C_VEL
LIN {X 0,Y 449.995,Z 137.434,A -85,B 0,C 180,E1 -8545.03,E2 -8545.03} C_VEL
LIN {X 0,Y 447.575,Z 137.734,A -85,B 0,C 180,E1 -8546,E2 -8546} C_VEL
LIN {X 0,Y 446.633,Z 137.854,A -85,B 0,C 180,E1 -8546.75,E2 -8546.75} C_VEL
LIN {X 0,Y 446.609,Z 137.853,A -85,B 0,C 180,E1 -8547.004,E2 -8547.004} C_VEL
LIN {X 0,Y 446.771,Z 137.994,A -85,B 0,C 180,E1 -8549.493,E2 -8549.493} C_VEL
LIN {X 0,Y 447.746,Z 145.333,A -85,B 0,C 180,E1 -8551.124,E2 -8551.124} C_VEL
LIN {X 0,Y 447.576,Z 151.153,A -85,B 0,C 180,E1 -8552.362,E2 -8552.362} C_VEL
LIN {X 0,Y 450.843,Z 167.969,A -85,B 0,C 180,E1 -8552.775,E2 -8552.775} C_VEL
LIN {X 0,Y 449.838,Z 258.728,A -85,B 0,C 180,E1 -8554.256,E2 -8554.256} C_VEL
LIN {X 0,Y 449.557,Z 272.499,A -85,B 0,C 180,E1 -8554.68,E2 -8554.68} C_VEL
LIN {X 0,Y 449.209,Z 285.368,A -85,B 0,C 180,E1 -8555.274,E2 -8555.274} C_VEL
LIN {X 0,Y 448.697,Z 297.951,A -85,B 0,C 180,E1 -8556.069,E2 -8556.069} C_VEL
LIN {X 0,Y 448.178,Z 309.162,A -85,B 0,C 180,E1 -8556.981,E2 -8556.981} C_VEL
LIN {X 0,Y 447.664,Z 318.256,A -85,B 0,C 180,E1 -8557.896,E2 -8557.896} C_VEL
LIN {X 0,Y 447.1,Z 327.577,A -85,B 0,C 180,E1 -8559.044,E2 -8559.044} C_VEL
LIN {X 0,Y 446.598,Z 336.619,A -85,B 0,C 180,E1 -8560.427,E2 -8560.427} C_VEL
LIN {X 0,Y 446.186,Z 343.891,A -85,B 0,C 180,E1 -8561.816,E2 -8561.816} C_VEL
LIN {X 0,Y 445.897,Z 349.664,A -85,B 0,C 180,E1 -8563.211,E2 -8563.211} C_VEL
LIN {X 0,Y 445.7,Z 354.201,A -85,B 0,C 180,E1 -8564.614,E2 -8564.614} C_VEL
LIN {X 0,Y 445.54,Z 357.175,A -85,B 0,C 180,E1 -8565.8,E2 -8565.8} C_VEL
LIN {X 0,Y 445.374,Z 360.011,A -85,B 0,C 180,E1 -8567.447,E2 -8567.447} C_VEL
LIN {X 0,Y 445.36,Z 361.329,A -85,B 0,C 180,E1 -8568.768,E2 -8568.768} C_VEL
LIN {X 0,Y 445.31,Z 361.778,A -85,B 0,C 180,E1 -8570.317,E2 -8570.317} C_VEL
LIN {X 0,Y 445.35,Z 361.411,A -85,B 0,C 180,E1 -8571.398,E2 -8571.398} C_VEL
LIN {X 0,Y 445.378,Z 360.737,A -85,B 0,C 180,E1 -8572.254,E2 -8572.254} C_VEL
LIN {X 0,Y 445.531,Z 358.566,A -85,B 0,C 180,E1 -8573.806,E2 -8573.806} C_VEL
LIN {X 0,Y 445.698,Z 355.569,A -85,B 0,C 180,E1 -8575.198,E2 -8575.198} C_VEL
LIN {X 0,Y 445.935,Z 351.144,A -85,B 0,C 180,E1 -8576.69,E2 -8576.69} C_VEL
LIN {X 0,Y 446.256,Z 345.288,A -85,B 0,C 180,E1 -8578.195,E2 -8578.195} C_VEL
LIN {X 0,Y 446.753,Z 337.779,A -85,B 0,C 180,E1 -8579.705,E2 -8579.705} C_VEL
LIN {X 0,Y 447.256,Z 329.854,A -85,B 0,C 180,E1 -8580.972,E2 -8580.972} C_VEL
LIN {X 0,Y 447.909,Z 320.024,A -85,B 0,C 180,E1 -8582.241,E2 -8582.241} C_VEL
LIN {X 0,Y 448.454,Z 310.254,A -85,B 0,C 180,E1 -8583.265,E2 -8583.265} C_VEL
LIN {X 0,Y 449.076,Z 299.636,A -85,B 0,C 180,E1 -8584.156,E2 -8584.156} C_VEL
LIN {X 0,Y 449.707,Z 286.939,A -85,B 0,C 180,E1 -8584.984,E2 -8584.984} C_VEL
LIN {X 0,Y 450.085,Z 274.546,A -85,B 0,C 180,E1 -8585.591,E2 -8585.591} C_VEL
LIN {X 0,Y 450.414,Z 261.336,A -85,B 0,C 180,E1 -8586.026,E2 -8586.026} C_VEL
LIN {X 0,Y 450.673,Z 242.717,A -85,B 0,C 180,E1 -8586.372,E2 -8586.372} C_VEL
LIN {X 0,Y 451.463,Z 167.618,A -85,B 0,C 180,E1 -8587.595,E2 -8587.595} C_VEL
LIN {X 0,Y 447.986,Z 151.535,A -85,B 0,C 180,E1 -8588.041,E2 -8588.041} C_VEL
LIN {X 0,Y 448.046,Z 146.391,A -85,B 0,C 180,E1 -8589.141,E2 -8589.141} C_VEL
LIN {X 0,Y 446.439,Z 137.877,A -85,B 0,C 180,E1 -8591.117,E2 -8591.117} C_VEL
LIN {X 0,Y 446.449,Z 137.876,A -85,B 0,C 180,E1 -8595.104,E2 -8595.104} C_VEL
LIN {X 0,Y 446.4,Z 137.882,A -85,B 0,C 180,E1 -8598.606,E2 -8598.606} C_VEL
LIN {X 0,Y 446.41,Z 137.877,A -85,B 0,C 180,E1 -8601.922,E2 -8601.922} C_VEL
LIN {X 0,Y 446.422,Z 137.876,A -85,B 0,C 180,E1 -8605.477,E2 -8605.477} C_VEL
LIN {X 0,Y 446.393,Z 137.883,A -85,B 0,C 180,E1 -8608.698,E2 -8608.698} C_VEL
LIN {X 0,Y 446.424,Z 137.874,A -85,B 0,C 180,E1 -8611.837,E2 -8611.837} C_VEL
LIN {X 0,Y 446.413,Z 137.88,A -85,B 0,C 180,E1 -8614.845,E2 -8614.845} C_VEL
LIN {X 0,Y 446.443,Z 137.871,A -85,B 0,C 180,E1 -8618.248,E2 -8618.248} C_VEL
LIN {X 0,Y 446.409,Z 137.872,A -85,B 0,C 180,E1 -8621.647,E2 -8621.647} C_VEL
LIN {X 0,Y 446.428,Z 137.873,A -85,B 0,C 180,E1 -8624.477,E2 -8624.477} C_VEL
LIN {X 0,Y 446.517,Z 137.862,A -85,B 0,C 180,E1 -8627.385,E2 -8627.385} C_VEL
LIN {X 0,Y 446.506,Z 137.863,A -85,B 0,C 180,E1 -8630.944,E2 -8630.944} C_VEL
LIN {X 0,Y 446.605,Z 137.848,A -85,B 0,C 180,E1 -8633.676,E2 -8633.676} C_VEL
LIN {X 0,Y 446.651,Z 137.843,A -85,B 0,C 180,E1 -8637.295,E2 -8637.295} C_VEL
LIN {X 0,Y 446.719,Z 137.842,A -85,B 0,C 180,E1 -8640,E2 -8640} C_VEL
LIN {X 0,Y 446.653,Z 137.838,A -85,B 0,C 180,E1 -8642.706,E2 -8642.706} C_VEL
LIN {X 0,Y 446.607,Z 137.849,A -85,B 0,C 180,E1 -8646.324,E2 -8646.324} C_VEL
LIN {X 0,Y 446.518,Z 137.859,A -85,B 0,C 180,E1 -8649.056,E2 -8649.056} C_VEL
LIN {X 0,Y 446.523,Z 137.856,A -85,B 0,C 180,E1 -8652.73,E2 -8652.73} C_VEL
LIN {X 0,Y 446.486,Z 137.864,A -85,B 0,C 180,E1 -8656.459,E2 -8656.459} C_VEL
LIN {X 0,Y 446.47,Z 137.871,A -85,B 0,C 180,E1 -8659.303,E2 -8659.303} C_VEL
LIN {X 0,Y 446.419,Z 137.867,A -85,B 0,C 180,E1 -8662.2,E2 -8662.2} C_VEL
LIN {X 0,Y 446.441,Z 137.874,A -85,B 0,C 180,E1 -8665.154,E2 -8665.154} C_VEL
LIN {X 0,Y 446.44,Z 137.871,A -85,B 0,C 180,E1 -8668.182,E2 -8668.182} C_VEL
LIN {X 0,Y 446.417,Z 137.877,A -85,B 0,C 180,E1 -8671.301,E2 -8671.301} C_VEL
LIN {X 0,Y 446.425,Z 137.874,A -85,B 0,C 180,E1 -8674.524,E2 -8674.524} C_VEL
LIN {X 0,Y 446.414,Z 137.874,A -85,B 0,C 180,E1 -8678.079,E2 -8678.079} C_VEL
LIN {X 0,Y 446.412,Z 137.877,A -85,B 0,C 180,E1 -8681.393,E2 -8681.393} C_VEL
LIN {X 0,Y 446.452,Z 137.872,A -85,B 0,C 180,E1 -8685.104,E2 -8685.104} C_VEL
LIN {X 0,Y 446.421,Z 137.881,A -85,B 0,C 180,E1 -8688.608,E2 -8688.608} C_VEL
LIN {X 0,Y 446.426,Z 137.875,A -85,B 0,C 180,E1 -8690.971,E2 -8690.971} C_VEL
LIN {X 0,Y 446.42,Z 137.877,A -85,B 0,C 180,E1 -8694.374,E2 -8694.374} C_VEL
LIN {X 0,Y 446.425,Z 137.877,A -85,B 0,C 180,E1 -8697.638,E2 -8697.638} C_VEL
LIN {X 0,Y 446.45,Z 137.874,A -85,B 0,C 180,E1 -8700.791,E2 -8700.791} C_VEL
LIN {X 0,Y 446.501,Z 137.957,A -85,B 0,C 180,E1 -8702.65,E2 -8702.65} C_VEL
LIN {X 0,Y 448.668,Z 148.352,A -85,B 0,C 180,E1 -8704.732,E2 -8704.732} C_VEL
LIN {X 0,Y 449.353,Z 152.713,A -85,B 0,C 180,E1 -8705.576,E2 -8705.576} C_VEL
LIN {X 0,Y 448.203,Z 172.443,A -85,B 0,C 180,E1 -8709.1,E2 -8709.1} C_VEL
LIN {X 0,Y 447.433,Z 188.838,A -85,B 0,C 180,E1 -8711.984,E2 -8711.984} C_VEL
LIN {X 0,Y 451.074,Z 212.258,A -85,B 0,C 180,E1 -8712.541,E2 -8712.541} C_VEL
LIN {X 0,Y 450.218,Z 298.445,A -85,B 0,C 180,E1 -8713.972,E2 -8713.972} C_VEL
LIN {X 0,Y 449.689,Z 312.126,A -85,B 0,C 180,E1 -8714.389,E2 -8714.389} C_VEL
LIN {X 0,Y 449.122,Z 324.963,A -85,B 0,C 180,E1 -8714.979,E2 -8714.979} C_VEL
LIN {X 0,Y 448.49,Z 336.7,A -85,B 0,C 180,E1 -8715.711,E2 -8715.711} C_VEL
LIN {X 0,Y 447.803,Z 348.654,A -85,B 0,C 180,E1 -8716.67,E2 -8716.67} C_VEL
LIN {X 0,Y 447.194,Z 359.274,A -85,B 0,C 180,E1 -8717.751,E2 -8717.751} C_VEL
LIN {X 0,Y 446.642,Z 368.332,A -85,B 0,C 180,E1 -8718.886,E2 -8718.886} C_VEL
LIN {X 0,Y 446.121,Z 377.194,A -85,B 0,C 180,E1 -8720.25,E2 -8720.25} C_VEL
LIN {X 0,Y 445.802,Z 384.321,A -85,B 0,C 180,E1 -8721.615,E2 -8721.615} C_VEL
LIN {X 0,Y 445.565,Z 390.84,A -85,B 0,C 180,E1 -8723.206,E2 -8723.206} C_VEL
LIN {X 0,Y 445.461,Z 395.151,A -85,B 0,C 180,E1 -8724.568,E2 -8724.568} C_VEL
LIN {X 0,Y 445.412,Z 397.439,A -85,B 0,C 180,E1 -8725.475,E2 -8725.475} C_VEL
LIN {X 0,Y 445.392,Z 399.27,A -85,B 0,C 180,E1 -8726.381,E2 -8726.381} C_VEL
LIN {X 0,Y 445.451,Z 400.655,A -85,B 0,C 180,E1 -8727.287,E2 -8727.287} C_VEL
LIN {X 0,Y 445.401,Z 402.233,A -85,B 0,C 180,E1 -8729.096,E2 -8729.096} C_VEL
LIN {X 0,Y 445.41,Z 402.411,A -85,B 0,C 180,E1 -8730,E2 -8730} C_VEL
LIN {X 0,Y 445.401,Z 402.167,A -85,B 0,C 180,E1 -8730.904,E2 -8730.904} C_VEL
LIN {X 0,Y 445.451,Z 400.514,A -85,B 0,C 180,E1 -8732.713,E2 -8732.713} C_VEL
LIN {X 0,Y 445.395,Z 399.055,A -85,B 0,C 180,E1 -8733.619,E2 -8733.619} C_VEL
LIN {X 0,Y 445.467,Z 396.053,A -85,B 0,C 180,E1 -8734.978,E2 -8734.978} C_VEL
LIN {X 0,Y 445.456,Z 391.981,A -85,B 0,C 180,E1 -8736.34,E2 -8736.34} C_VEL
LIN {X 0,Y 445.699,Z 385.724,A -85,B 0,C 180,E1 -8737.93,E2 -8737.93} C_VEL
LIN {X 0,Y 445.943,Z 378.902,A -85,B 0,C 180,E1 -8739.296,E2 -8739.296} C_VEL
LIN {X 0,Y 446.365,Z 370.422,A -85,B 0,C 180,E1 -8740.661,E2 -8740.661} C_VEL
LIN {X 0,Y 446.89,Z 361.685,A -85,B 0,C 180,E1 -8741.797,E2 -8741.797} C_VEL
LIN {X 0,Y 447.372,Z 351.963,A -85,B 0,C 180,E1 -8742.834,E2 -8742.834} C_VEL
LIN {X 0,Y 447.935,Z 341.66,A -85,B 0,C 180,E1 -8743.728,E2 -8743.728} C_VEL
LIN {X 0,Y 448.498,Z 330.2,A -85,B 0,C 180,E1 -8744.52,E2 -8744.52} C_VEL
LIN {X 0,Y 449.003,Z 318.364,A -85,B 0,C 180,E1 -8745.141,E2 -8745.141} C_VEL
LIN {X 0,Y 449.55,Z 304.73,A -85,B 0,C 180,E1 -8745.645,E2 -8745.645} C_VEL
LIN {X 0,Y 449.804,Z 292.577,A -85,B 0,C 180,E1 -8745.926,E2 -8745.926} C_VEL
LIN {X 0,Y 450.447,Z 211.696,A -85,B 0,C 180,E1 -8747.231,E2 -8747.231} C_VEL
LIN {X 0,Y 447.257,Z 189.2,A -85,B 0,C 180,E1 -8747.737,E2 -8747.737} C_VEL
LIN {X 0,Y 448.012,Z 171.01,A -85,B 0,C 180,E1 -8750.909,E2 -8750.909} C_VEL
LIN {X 0,Y 448.929,Z 153.378,A -85,B 0,C 180,E1 -8754.018,E2 -8754.018} C_VEL
LIN {X 0,Y 448.762,Z 149.5,A -85,B 0,C 180,E1 -8754.724,E2 -8754.724} C_VEL
LIN {X 0,Y 446.524,Z 137.864,A -85,B 0,C 180,E1 -8756.99,E2 -8756.99} C_VEL
LIN {X 0,Y 446.429,Z 137.879,A -85,B 0,C 180,E1 -8760.249,E2 -8760.249} C_VEL
LIN {X 0,Y 446.447,Z 137.871,A -85,B 0,C 180,E1 -8763.453,E2 -8763.453} C_VEL
LIN {X 0,Y 446.403,Z 137.875,A -85,B 0,C 180,E1 -8766.745,E2 -8766.745} C_VEL
LIN {X 0,Y 446.479,Z 137.869,A -85,B 0,C 180,E1 -8769.528,E2 -8769.528} C_VEL
LIN {X 0,Y 446.43,Z 137.872,A -85,B 0,C 180,E1 -8772.604,E2 -8772.604} C_VEL
LIN {X 0,Y 446.452,Z 137.87,A -85,B 0,C 180,E1 -8775.103,E2 -8775.103} C_VEL
LIN {X 0,Y 446.429,Z 137.872,A -85,B 0,C 180,E1 -8778.609,E2 -8778.609} C_VEL
LIN {X 0,Y 446.438,Z 137.872,A -85,B 0,C 180,E1 -8780.972,E2 -8780.972} C_VEL
LIN {X 0,Y 446.418,Z 137.873,A -85,B 0,C 180,E1 -8784.374,E2 -8784.374} C_VEL
LIN {X 0,Y 446.42,Z 137.878,A -85,B 0,C 180,E1 -8787.638,E2 -8787.638} C_VEL
LIN {X 0,Y 446.448,Z 137.871,A -85,B 0,C 180,E1 -8790.79,E2 -8790.79} C_VEL
LIN {X 0,Y 446.478,Z 137.867,A -85,B 0,C 180,E1 -8793.848,E2 -8793.848} C_VEL
LIN {X 0,Y 446.429,Z 137.875,A -85,B 0,C 180,E1 -8796.823,E2 -8796.823} C_VEL
LIN {X 0,Y 446.444,Z 137.871,A -85,B 0,C 180,E1 -8799.737,E2 -8799.737} C_VEL
LIN {X 0,Y 446.457,Z 137.87,A -85,B 0,C 180,E1 -8802.597,E2 -8802.597} C_VEL
LIN {X 0,Y 446.47,Z 137.869,A -85,B 0,C 180,E1 -8805.412,E2 -8805.412} C_VEL
LIN {X 0,Y 446.517,Z 137.861,A -85,B 0,C 180,E1 -8808.193,E2 -8808.193} C_VEL
LIN {X 0,Y 446.532,Z 137.866,A -85,B 0,C 180,E1 -8810.944,E2 -8810.944} C_VEL
LIN {X 0,Y 446.621,Z 137.848,A -85,B 0,C 180,E1 -8813.676,E2 -8813.676} C_VEL
LIN {X 0,Y 446.691,Z 137.841,A -85,B 0,C 180,E1 -8817.294,E2 -8817.294} C_VEL
LIN {X 0,Y 446.793,Z 137.827,A -85,B 0,C 180,E1 -8820,E2 -8820} C_VEL
LIN {X 0,Y 446.707,Z 137.844,A -85,B 0,C 180,E1 -8822.705,E2 -8822.705} C_VEL
LIN {X 0,Y 446.639,Z 137.85,A -85,B 0,C 180,E1 -8826.324,E2 -8826.324} C_VEL
LIN {X 0,Y 446.536,Z 137.86,A -85,B 0,C 180,E1 -8829.055,E2 -8829.055} C_VEL
LIN {X 0,Y 446.521,Z 137.864,A -85,B 0,C 180,E1 -8832.73,E2 -8832.73} C_VEL
LIN {X 0,Y 446.495,Z 137.87,A -85,B 0,C 180,E1 -8836.227,E2 -8836.227} C_VEL
LIN {X 0,Y 446.468,Z 137.867,A -85,B 0,C 180,E1 -8839.303,E2 -8839.303} C_VEL
LIN {X 0,Y 446.418,Z 137.881,A -85,B 0,C 180,E1 -8842.199,E2 -8842.199} C_VEL
LIN {X 0,Y 446.443,Z 137.87,A -85,B 0,C 180,E1 -8845.153,E2 -8845.153} C_VEL
LIN {X 0,Y 446.484,Z 137.871,A -85,B 0,C 180,E1 -8848.179,E2 -8848.179} C_VEL
LIN {X 0,Y 446.418,Z 137.878,A -85,B 0,C 180,E1 -8851.775,E2 -8851.775} C_VEL
LIN {X 0,Y 446.428,Z 137.873,A -85,B 0,C 180,E1 -8854.523,E2 -8854.523} C_VEL
LIN {X 0,Y 446.415,Z 137.878,A -85,B 0,C 180,E1 -8858.079,E2 -8858.079} C_VEL
LIN {X 0,Y 446.426,Z 137.872,A -85,B 0,C 180,E1 -8860.918,E2 -8860.918} C_VEL
LIN {X 0,Y 446.399,Z 137.881,A -85,B 0,C 180,E1 -8863.846,E2 -8863.846} C_VEL
LIN {X 0,Y 446.397,Z 137.876,A -85,B 0,C 180,E1 -8866.404,E2 -8866.404} C_VEL
LIN {X 0,Y 446.425,Z 137.874,A -85,B 0,C 180,E1 -8869.083,E2 -8869.083} C_VEL
LIN {X 0,Y 446.406,Z 137.875,A -85,B 0,C 180,E1 -8872.121,E2 -8872.121} C_VEL
LIN {X 0,Y 446.422,Z 137.88,A -85,B 0,C 180,E1 -8875.477,E2 -8875.477} C_VEL
LIN {X 0,Y 446.414,Z 137.874,A -85,B 0,C 180,E1 -8878.7,E2 -8878.7} C_VEL
LIN {X 0,Y 446.484,Z 137.866,A -85,B 0,C 180,E1 -8881.822,E2 -8881.822} C_VEL
LIN {X 0,Y 446.449,Z 137.872,A -85,B 0,C 180,E1 -8884.847,E2 -8884.847} C_VEL
LIN {X 0,Y 446.448,Z 137.869,A -85,B 0,C 180,E1 -8888.245,E2 -8888.245} C_VEL
LIN {X 0,Y 446.451,Z 137.87,A -85,B 0,C 180,E1 -8891.649,E2 -8891.649} C_VEL
LIN {X 0,Y 446.507,Z 137.864,A -85,B 0,C 180,E1 -8894.48,E2 -8894.48} C_VEL
LIN {X 0,Y 446.517,Z 137.861,A -85,B 0,C 180,E1 -8898.193,E2 -8898.193} C_VEL
LIN {X 0,Y 446.532,Z 137.865,A -85,B 0,C 180,E1 -8900.945,E2 -8900.945} C_VEL
LIN {X 0,Y 446.621,Z 137.848,A -85,B 0,C 180,E1 -8903.676,E2 -8903.676} C_VEL
LIN {X 0,Y 446.609,Z 137.853,A -85,B 0,C 180,E1 -8907.004,E2 -8907.004} C_VEL
LIN {X 0,Y 446.01,Z 137.953,A -85,B 0,C 180,E1 -8907.523,E2 -8907.523} C_VEL
LIN {X 0,Y 443.157,Z 138.286,A -85,B 0,C 180,E1 -8908.338,E2 -8908.338} C_VEL
LIN {X 0,Y 440.429,Z 138.788,A -85,B 0,C 180,E1 -8909.131,E2 -8909.131} C_VEL
LIN {X 0,Y 439.929,Z 139.924,A -85,B 0,C 180,E1 -8909.566,E2 -8909.566} C_VEL
LIN {X 0,Y 439.948,Z 140.079,A -85,B 0,C 180,E1 -8909.603,E2 -8909.603} C_VEL
LIN {X 0,Y 440.791,Z 146.94,A -85,B 0,C 180,E1 -8911.142,E2 -8911.142} C_VEL
LIN {X 0,Y 440.638,Z 151.452,A -85,B 0,C 180,E1 -8912.114,E2 -8912.114} C_VEL
LIN {X 0,Y 444.001,Z 168.494,A -85,B 0,C 180,E1 -8912.535,E2 -8912.535} C_VEL
LIN {X 0,Y 442.975,Z 259.08,A -85,B 0,C 180,E1 -8914.037,E2 -8914.037} C_VEL
LIN {X 0,Y 442.689,Z 272.09,A -85,B 0,C 180,E1 -8914.439,E2 -8914.439} C_VEL
LIN {X 0,Y 442.337,Z 284.662,A -85,B 0,C 180,E1 -8915.013,E2 -8915.013} C_VEL
LIN {X 0,Y 441.868,Z 295.91,A -85,B 0,C 180,E1 -8915.705,E2 -8915.705} C_VEL
LIN {X 0,Y 441.356,Z 307.53,A -85,B 0,C 180,E1 -8916.63,E2 -8916.63} C_VEL
LIN {X 0,Y 440.72,Z 318.053,A -85,B 0,C 180,E1 -8917.675,E2 -8917.675} C_VEL
LIN {X 0,Y 440.188,Z 326.639,A -85,B 0,C 180,E1 -8918.724,E2 -8918.724} C_VEL
LIN {X 0,Y 439.707,Z 334.542,A -85,B 0,C 180,E1 -8919.894,E2 -8919.894} C_VEL
LIN {X 0,Y 439.269,Z 342.243,A -85,B 0,C 180,E1 -8921.303,E2 -8921.303} C_VEL
LIN {X 0,Y 438.891,Z 349.359,A -85,B 0,C 180,E1 -8922.955,E2 -8922.955} C_VEL
LIN {X 0,Y 438.639,Z 354.056,A -85,B 0,C 180,E1 -8924.38,E2 -8924.38} C_VEL
LIN {X 0,Y 438.451,Z 357.78,A -85,B 0,C 180,E1 -8925.899,E2 -8925.899} C_VEL
LIN {X 0,Y 438.273,Z 360.712,A -85,B 0,C 180,E1 -8927.739,E2 -8927.739} C_VEL
LIN {X 0,Y 438.263,Z 361.717,A -85,B 0,C 180,E1 -8928.893,E2 -8928.893} C_VEL
LIN {X 0,Y 438.238,Z 362.052,A -85,B 0,C 180,E1 -8930.66,E2 -8930.66} C_VEL
LIN {X 0,Y 438.263,Z 361.631,A -85,B 0,C 180,E1 -8931.644,E2 -8931.644} C_VEL
LIN {X 0,Y 438.327,Z 360.706,A -85,B 0,C 180,E1 -8932.632,E2 -8932.632} C_VEL
LIN {X 0,Y 438.47,Z 358.712,A -85,B 0,C 180,E1 -8933.99,E2 -8933.99} C_VEL
LIN {X 0,Y 438.724,Z 355.053,A -85,B 0,C 180,E1 -8935.628,E2 -8935.628} C_VEL
LIN {X 0,Y 438.977,Z 350.361,A -85,B 0,C 180,E1 -8937.148,E2 -8937.148} C_VEL
LIN {X 0,Y 439.351,Z 344.203,A -85,B 0,C 180,E1 -8938.678,E2 -8938.678} C_VEL
LIN {X 0,Y 439.85,Z 337.181,A -85,B 0,C 180,E1 -8940.05,E2 -8940.05} C_VEL
LIN {X 0,Y 440.356,Z 329.696,A -85,B 0,C 180,E1 -8941.245,E2 -8941.245} C_VEL
LIN {X 0,Y 441.042,Z 320.076,A -85,B 0,C 180,E1 -8942.496,E2 -8942.496} C_VEL
LIN {X 0,Y 441.661,Z 309.858,A -85,B 0,C 180,E1 -8943.571,E2 -8943.571} C_VEL
LIN {X 0,Y 442.319,Z 299.138,A -85,B 0,C 180,E1 -8944.467,E2 -8944.467} C_VEL
LIN {X 0,Y 442.938,Z 287.196,A -85,B 0,C 180,E1 -8945.251,E2 -8945.251} C_VEL
LIN {X 0,Y 443.318,Z 275.3,A -85,B 0,C 180,E1 -8945.844,E2 -8945.844} C_VEL
LIN {X 0,Y 443.686,Z 262.094,A -85,B 0,C 180,E1 -8946.292,E2 -8946.292} C_VEL
LIN {X 0,Y 443.933,Z 244.208,A -85,B 0,C 180,E1 -8946.636,E2 -8946.636} C_VEL
LIN {X 0,Y 444.738,Z 168.339,A -85,B 0,C 180,E1 -8947.893,E2 -8947.893} C_VEL
LIN {X 0,Y 441.129,Z 151.818,A -85,B 0,C 180,E1 -8948.366,E2 -8948.366} C_VEL
LIN {X 0,Y 441.071,Z 147.38,A -85,B 0,C 180,E1 -8949.342,E2 -8949.342} C_VEL
LIN {X 0,Y 439.379,Z 138.757,A -85,B 0,C 180,E1 -8951.373,E2 -8951.373} C_VEL
LIN {X 0,Y 439.397,Z 138.755,A -85,B 0,C 180,E1 -8954.73,E2 -8954.73} C_VEL
LIN {X 0,Y 439.348,Z 138.76,A -85,B 0,C 180,E1 -8957.79,E2 -8957.79} C_VEL
LIN {X 0,Y 439.362,Z 138.759,A -85,B 0,C 180,E1 -8961.403,E2 -8961.403} C_VEL
LIN {X 0,Y 439.395,Z 138.752,A -85,B 0,C 180,E1 -8964.844,E2 -8964.844} C_VEL
LIN {X 0,Y 439.354,Z 138.757,A -85,B 0,C 180,E1 -8968.138,E2 -8968.138} C_VEL
LIN {X 0,Y 439.38,Z 138.753,A -85,B 0,C 180,E1 -8971.324,E2 -8971.324} C_VEL
LIN {X 0,Y 439.354,Z 138.758,A -85,B 0,C 180,E1 -8974.412,E2 -8974.412} C_VEL
LIN {X 0,Y 439.352,Z 138.751,A -85,B 0,C 180,E1 -8977.424,E2 -8977.424} C_VEL
LIN {X 0,Y 439.381,Z 138.751,A -85,B 0,C 180,E1 -8980.686,E2 -8980.686} C_VEL
LIN {X 0,Y 439.401,Z 138.751,A -85,B 0,C 180,E1 -8984.222,E2 -8984.222} C_VEL
LIN {X 0,Y 439.466,Z 138.74,A -85,B 0,C 180,E1 -8987.297,E2 -8987.297} C_VEL
LIN {X 0,Y 439.473,Z 138.74,A -85,B 0,C 180,E1 -8990.798,E2 -8990.798} C_VEL
LIN {X 0,Y 439.558,Z 138.726,A -85,B 0,C 180,E1 -8993.574,E2 -8993.574} C_VEL
LIN {X 0,Y 439.401,Z 138.748,A -85,B 0,C 180,E1 -8995.413,E2 -8995.413} C_VEL
LIN {X 0,Y 439.626,Z 138.718,A -85,B 0,C 180,E1 -8998.168,E2 -8998.168} C_VEL
LIN {X 0,Y 439.67,Z 138.72,A -85,B 0,C 180,E1 -9000,E2 -9000} C_VEL
LIN {X 0,Y 439.604,Z 138.715,A -85,B 0,C 180,E1 -9002.749,E2 -9002.749} C_VEL
LIN {X 0,Y 439.56,Z 138.727,A -85,B 0,C 180,E1 -9006.426,E2 -9006.426} C_VEL
LIN {X 0,Y 439.485,Z 138.737,A -85,B 0,C 180,E1 -9009.202,E2 -9009.202} C_VEL
LIN {X 0,Y 439.467,Z 138.736,A -85,B 0,C 180,E1 -9012.938,E2 -9012.938} C_VEL
LIN {X 0,Y 439.446,Z 138.741,A -85,B 0,C 180,E1 -9016.347,E2 -9016.347} C_VEL
LIN {X 0,Y 439.404,Z 138.75,A -85,B 0,C 180,E1 -9019.626,E2 -9019.626} C_VEL
LIN {X 0,Y 439.365,Z 138.747,A -85,B 0,C 180,E1 -9022.576,E2 -9022.576} C_VEL
LIN {X 0,Y 439.378,Z 138.749,A -85,B 0,C 180,E1 -9025.587,E2 -9025.587} C_VEL
LIN {X 0,Y 439.393,Z 138.752,A -85,B 0,C 180,E1 -9028.675,E2 -9028.675} C_VEL
LIN {X 0,Y 439.37,Z 138.752,A -85,B 0,C 180,E1 -9032.03,E2 -9032.03} C_VEL
LIN {X 0,Y 439.394,Z 138.751,A -85,B 0,C 180,E1 -9035.34,E2 -9035.34} C_VEL
LIN {X 0,Y 439.37,Z 138.757,A -85,B 0,C 180,E1 -9038.597,E2 -9038.597} C_VEL
LIN {X 0,Y 439.372,Z 138.755,A -85,B 0,C 180,E1 -9041.254,E2 -9041.254} C_VEL
LIN {X 0,Y 439.401,Z 138.754,A -85,B 0,C 180,E1 -9044.73,E2 -9044.73} C_VEL
LIN {X 0,Y 439.386,Z 138.754,A -85,B 0,C 180,E1 -9047.794,E2 -9047.794} C_VEL
LIN {X 0,Y 439.391,Z 138.755,A -85,B 0,C 180,E1 -9050.223,E2 -9050.223} C_VEL
LIN {X 0,Y 439.374,Z 138.754,A -85,B 0,C 180,E1 -9053.713,E2 -9053.713} C_VEL
LIN {X 0,Y 439.375,Z 138.755,A -85,B 0,C 180,E1 -9057.054,E2 -9057.054} C_VEL
LIN {X 0,Y 439.384,Z 138.756,A -85,B 0,C 180,E1 -9060.274,E2 -9060.274} C_VEL
LIN {X 0,Y 439.488,Z 138.858,A -85,B 0,C 180,E1 -9062.371,E2 -9062.371} C_VEL
LIN {X 0,Y 442.006,Z 151.053,A -85,B 0,C 180,E1 -9064.851,E2 -9064.851} C_VEL
LIN {X 0,Y 442.392,Z 154.945,A -85,B 0,C 180,E1 -9065.604,E2 -9065.604} C_VEL
LIN {X 0,Y 441.249,Z 173.632,A -85,B 0,C 180,E1 -9069,E2 -9069} C_VEL
LIN {X 0,Y 440.537,Z 188.546,A -85,B 0,C 180,E1 -9071.662,E2 -9071.662} C_VEL
LIN {X 0,Y 444.004,Z 210.623,A -85,B 0,C 180,E1 -9072.201,E2 -9072.201} C_VEL
LIN {X 0,Y 444.323,Z 215.06,A -85,B 0,C 180,E1 -9072.291,E2 -9072.291} C_VEL
LIN {X 0,Y 443.481,Z 298.088,A -85,B 0,C 180,E1 -9073.692,E2 -9073.692} C_VEL
LIN {X 0,Y 442.937,Z 311.018,A -85,B 0,C 180,E1 -9074.086,E2 -9074.086} C_VEL
LIN {X 0,Y 442.35,Z 324.111,A -85,B 0,C 180,E1 -9074.684,E2 -9074.684} C_VEL
LIN {X 0,Y 441.606,Z 336.752,A -85,B 0,C 180,E1 -9075.484,E2 -9075.484} C_VEL
LIN {X 0,Y 440.952,Z 347.413,A -85,B 0,C 180,E1 -9076.348,E2 -9076.348} C_VEL
LIN {X 0,Y 440.274,Z 358.2,A -85,B 0,C 180,E1 -9077.438,E2 -9077.438} C_VEL
LIN {X 0,Y 439.666,Z 368.199,A -85,B 0,C 180,E1 -9078.708,E2 -9078.708} C_VEL
LIN {X 0,Y 439.087,Z 377.026,A -85,B 0,C 180,E1 -9080.092,E2 -9080.092} C_VEL
LIN {X 0,Y 438.763,Z 384.101,A -85,B 0,C 180,E1 -9081.479,E2 -9081.479} C_VEL
LIN {X 0,Y 438.496,Z 390.589,A -85,B 0,C 180,E1 -9083.096,E2 -9083.096} C_VEL
LIN {X 0,Y 438.358,Z 394.876,A -85,B 0,C 180,E1 -9084.48,E2 -9084.48} C_VEL
LIN {X 0,Y 438.34,Z 397.157,A -85,B 0,C 180,E1 -9085.402,E2 -9085.402} C_VEL
LIN {X 0,Y 438.292,Z 398.971,A -85,B 0,C 180,E1 -9086.322,E2 -9086.322} C_VEL
LIN {X 0,Y 438.375,Z 400.351,A -85,B 0,C 180,E1 -9087.243,E2 -9087.243} C_VEL
LIN {X 0,Y 438.311,Z 401.918,A -85,B 0,C 180,E1 -9089.081,E2 -9089.081} C_VEL
LIN {X 0,Y 438.318,Z 402.084,A -85,B 0,C 180,E1 -9090,E2 -9090} C_VEL
LIN {X 0,Y 438.32,Z 401.197,A -85,B 0,C 180,E1 -9091.838,E2 -9091.838} C_VEL
LIN {X 0,Y 438.376,Z 400.169,A -85,B 0,C 180,E1 -9092.757,E2 -9092.757} C_VEL
LIN {X 0,Y 438.297,Z 398.696,A -85,B 0,C 180,E1 -9093.677,E2 -9093.677} C_VEL
LIN {X 0,Y 438.374,Z 395.68,A -85,B 0,C 180,E1 -9095.059,E2 -9095.059} C_VEL
LIN {X 0,Y 438.369,Z 391.593,A -85,B 0,C 180,E1 -9096.443,E2 -9096.443} C_VEL
LIN {X 0,Y 438.626,Z 385.311,A -85,B 0,C 180,E1 -9098.059,E2 -9098.059} C_VEL
LIN {X 0,Y 438.886,Z 378.458,A -85,B 0,C 180,E1 -9099.447,E2 -9099.447} C_VEL
LIN {X 0,Y 439.354,Z 369.927,A -85,B 0,C 180,E1 -9100.833,E2 -9100.833} C_VEL
LIN {X 0,Y 439.88,Z 361.139,A -85,B 0,C 180,E1 -9101.988,E2 -9101.988} C_VEL
LIN {X 0,Y 440.409,Z 351.023,A -85,B 0,C 180,E1 -9103.073,E2 -9103.073} C_VEL
LIN {X 0,Y 441.079,Z 339.512,A -85,B 0,C 180,E1 -9104.063,E2 -9104.063} C_VEL
LIN {X 0,Y 441.707,Z 327.383,A -85,B 0,C 180,E1 -9104.866,E2 -9104.866} C_VEL
LIN {X 0,Y 442.257,Z 314.731,A -85,B 0,C 180,E1 -9105.496,E2 -9105.496} C_VEL
LIN {X 0,Y 442.729,Z 302.444,A -85,B 0,C 180,E1 -9105.922,E2 -9105.922} C_VEL
LIN {X 0,Y 443.003,Z 286.876,A -85,B 0,C 180,E1 -9106.237,E2 -9106.237} C_VEL
LIN {X 0,Y 443.615,Z 212.601,A -85,B 0,C 180,E1 -9107.453,E2 -9107.453} C_VEL
LIN {X 0,Y 440.258,Z 188.989,A -85,B 0,C 180,E1 -9107.98,E2 -9107.98} C_VEL
LIN {X 0,Y 441.116,Z 170.543,A -85,B 0,C 180,E1 -9111.251,E2 -9111.251} C_VEL
LIN {X 0,Y 442.034,Z 152.85,A -85,B 0,C 180,E1 -9114.417,E2 -9114.417} C_VEL
LIN {X 0,Y 440.063,Z 141.645,A -85,B 0,C 180,E1 -9116.575,E2 -9116.575} C_VEL
LIN {X 0,Y 439.465,Z 138.744,A -85,B 0,C 180,E1 -9117.179,E2 -9117.179} C_VEL
LIN {X 0,Y 439.382,Z 138.757,A -85,B 0,C 180,E1 -9120.26,E2 -9120.26} C_VEL
LIN {X 0,Y 439.398,Z 138.752,A -85,B 0,C 180,E1 -9123.724,E2 -9123.724} C_VEL
LIN {X 0,Y 439.349,Z 138.753,A -85,B 0,C 180,E1 -9126.887,E2 -9126.887} C_VEL
LIN {X 0,Y 439.414,Z 138.753,A -85,B 0,C 180,E1 -9129.851,E2 -9129.851} C_VEL
LIN {X 0,Y 439.382,Z 138.749,A -85,B 0,C 180,E1 -9132.627,E2 -9132.627} C_VEL
LIN {X 0,Y 439.4,Z 138.75,A -85,B 0,C 180,E1 -9135.27,E2 -9135.27} C_VEL
LIN {X 0,Y 439.389,Z 138.749,A -85,B 0,C 180,E1 -9138.743,E2 -9138.743} C_VEL
LIN {X 0,Y 439.372,Z 138.758,A -85,B 0,C 180,E1 -9141.608,E2 -9141.608} C_VEL
LIN {X 0,Y 439.397,Z 138.749,A -85,B 0,C 180,E1 -9144.844,E2 -9144.844} C_VEL
LIN {X 0,Y 439.372,Z 138.751,A -85,B 0,C 180,E1 -9148.139,E2 -9148.139} C_VEL
LIN {X 0,Y 439.433,Z 138.747,A -85,B 0,C 180,E1 -9151.598,E2 -9151.598} C_VEL
LIN {X 0,Y 439.401,Z 138.747,A -85,B 0,C 180,E1 -9154.415,E2 -9154.415} C_VEL
LIN {X 0,Y 439.365,Z 138.756,A -85,B 0,C 180,E1 -9157.424,E2 -9157.424} C_VEL
LIN {X 0,Y 439.441,Z 138.744,A -85,B 0,C 180,E1 -9160.663,E2 -9160.663} C_VEL
LIN {X 0,Y 439.462,Z 138.74,A -85,B 0,C 180,E1 -9164.224,E2 -9164.224} C_VEL
LIN {X 0,Y 439.483,Z 138.737,A -85,B 0,C 180,E1 -9168.001,E2 -9168.001} C_VEL
LIN {X 0,Y 439.503,Z 138.734,A -85,B 0,C 180,E1 -9171.725,E2 -9171.725} C_VEL
LIN {X 0,Y 439.611,Z 138.725,A -85,B 0,C 180,E1 -9174.495,E2 -9174.495} C_VEL
LIN {X 0,Y 439.635,Z 138.719,A -85,B 0,C 180,E1 -9178.168,E2 -9178.168} C_VEL
LIN {X 0,Y 439.762,Z 138.703,A -85,B 0,C 180,E1 -9180,E2 -9180} C_VEL
LIN {X 0,Y 439.654,Z 138.722,A -85,B 0,C 180,E1 -9182.749,E2 -9182.749} C_VEL
LIN {X 0,Y 439.611,Z 138.727,A -85,B 0,C 180,E1 -9186.425,E2 -9186.425} C_VEL
LIN {X 0,Y 439.498,Z 138.735,A -85,B 0,C 180,E1 -9189.201,E2 -9189.201} C_VEL
LIN {X 0,Y 439.465,Z 138.741,A -85,B 0,C 180,E1 -9192.937,E2 -9192.937} C_VEL
LIN {X 0,Y 439.446,Z 138.749,A -85,B 0,C 180,E1 -9196.348,E2 -9196.348} C_VEL
LIN {X 0,Y 439.401,Z 138.748,A -85,B 0,C 180,E1 -9199.626,E2 -9199.626} C_VEL
LIN {X 0,Y 439.363,Z 138.755,A -85,B 0,C 180,E1 -9202.575,E2 -9202.575} C_VEL
LIN {X 0,Y 439.397,Z 138.749,A -85,B 0,C 180,E1 -9205.585,E2 -9205.585} C_VEL
LIN {X 0,Y 439.416,Z 138.746,A -85,B 0,C 180,E1 -9208.673,E2 -9208.673} C_VEL
LIN {X 0,Y 439.369,Z 138.758,A -85,B 0,C 180,E1 -9212.03,E2 -9212.03} C_VEL
LIN {X 0,Y 439.393,Z 138.75,A -85,B 0,C 180,E1 -9215.34,E2 -9215.34} C_VEL
LIN {X 0,Y 439.384,Z 138.749,A -85,B 0,C 180,E1 -9218.595,E2 -9218.595} C_VEL
LIN {X 0,Y 439.387,Z 138.751,A -85,B 0,C 180,E1 -9221.257,E2 -9221.257} C_VEL
LIN {X 0,Y 439.399,Z 138.747,A -85,B 0,C 180,E1 -9224.729,E2 -9224.729} C_VEL
LIN {X 0,Y 439.395,Z 138.753,A -85,B 0,C 180,E1 -9227.796,E2 -9227.796} C_VEL
LIN {X 0,Y 439.393,Z 138.749,A -85,B 0,C 180,E1 -9230.224,E2 -9230.224} C_VEL
LIN {X 0,Y 439.372,Z 138.755,A -85,B 0,C 180,E1 -9233.713,E2 -9233.713} C_VEL
LIN {X 0,Y 439.371,Z 138.754,A -85,B 0,C 180,E1 -9237.054,E2 -9237.054} C_VEL
LIN {X 0,Y 439.381,Z 138.75,A -85,B 0,C 180,E1 -9240.274,E2 -9240.274} C_VEL
LIN {X 0,Y 439.428,Z 138.749,A -85,B 0,C 180,E1 -9243.396,E2 -9243.396} C_VEL
LIN {X 0,Y 439.385,Z 138.749,A -85,B 0,C 180,E1 -9246.43,E2 -9246.43} C_VEL
LIN {X 0,Y 439.388,Z 138.753,A -85,B 0,C 180,E1 -9249.397,E2 -9249.397} C_VEL
LIN {X 0,Y 439.405,Z 138.747,A -85,B 0,C 180,E1 -9252.309,E2 -9252.309} C_VEL
LIN {X 0,Y 439.447,Z 138.746,A -85,B 0,C 180,E1 -9255.174,E2 -9255.174} C_VEL
LIN {X 0,Y 439.483,Z 138.737,A -85,B 0,C 180,E1 -9258.001,E2 -9258.001} C_VEL
LIN {X 0,Y 439.503,Z 138.734,A -85,B 0,C 180,E1 -9261.726,E2 -9261.726} C_VEL
LIN {X 0,Y 439.611,Z 138.725,A -85,B 0,C 180,E1 -9264.496,E2 -9264.496} C_VEL
LIN {X 0,Y 439.635,Z 138.724,A -85,B 0,C 180,E1 -9268.168,E2 -9268.168} C_VEL
LIN {X 0,Y 439.693,Z 138.829,A -85,B 0,C 180,E1 -9269.313,E2 -9269.313} C_VEL
LIN {X 0,Y 439.948,Z 140.079,A -85,B 0,C 180,E1 -9269.603,E2 -9269.603} C_VEL
LIN {X 0,Y 439.562,Z 142.158,A -85,B 0,C 180,E1 -9270.038,E2 -9270.038} C_VEL
LIN {X 0,Y 437.076,Z 145.753,A -85,B 0,C 180,E1 -9270.702,E2 -9270.702} C_VEL
LIN {X 0,Y 434.38,Z 149.409,A -85,B 0,C 180,E1 -9271.37,E2 -9271.37} C_VEL
LIN {X 0,Y 433.7,Z 151.548,A -85,B 0,C 180,E1 -9271.81,E2 -9271.81} C_VEL
LIN {X 0,Y 433.799,Z 152.43,A -85,B 0,C 180,E1 -9271.872,E2 -9271.872} C_VEL
LIN {X 0,Y 437.163,Z 169.991,A -85,B 0,C 180,E1 -9272.303,E2 -9272.303} C_VEL
LIN {X 0,Y 436.124,Z 259.423,A -85,B 0,C 180,E1 -9273.812,E2 -9273.812} C_VEL
LIN {X 0,Y 435.82,Z 272.429,A -85,B 0,C 180,E1 -9274.219,E2 -9274.219} C_VEL
LIN {X 0,Y 435.441,Z 285.003,A -85,B 0,C 180,E1 -9274.803,E2 -9274.803} C_VEL
LIN {X 0,Y 434.925,Z 297.03,A -85,B 0,C 180,E1 -9275.564,E2 -9275.564} C_VEL
LIN {X 0,Y 434.368,Z 308.518,A -85,B 0,C 180,E1 -9276.503,E2 -9276.503} C_VEL
LIN {X 0,Y 433.773,Z 317.848,A -85,B 0,C 180,E1 -9277.448,E2 -9277.448} C_VEL
LIN {X 0,Y 433.159,Z 327.409,A -85,B 0,C 180,E1 -9278.632,E2 -9278.632} C_VEL
LIN {X 0,Y 432.578,Z 336.595,A -85,B 0,C 180,E1 -9280.059,E2 -9280.059} C_VEL
LIN {X 0,Y 432.149,Z 343.995,A -85,B 0,C 180,E1 -9281.492,E2 -9281.492} C_VEL
LIN {X 0,Y 431.849,Z 349.093,A -85,B 0,C 180,E1 -9282.717,E2 -9282.717} C_VEL
LIN {X 0,Y 431.61,Z 353.842,A -85,B 0,C 180,E1 -9284.138,E2 -9284.138} C_VEL
LIN {X 0,Y 431.479,Z 356.434,A -85,B 0,C 180,E1 -9285.106,E2 -9285.106} C_VEL
LIN {X 0,Y 431.354,Z 358.521,A -85,B 0,C 180,E1 -9286.08,E2 -9286.08} C_VEL
LIN {X 0,Y 431.221,Z 360.18,A -85,B 0,C 180,E1 -9287.06,E2 -9287.06} C_VEL
LIN {X 0,Y 431.197,Z 361.371,A -85,B 0,C 180,E1 -9288.04,E2 -9288.04} C_VEL
LIN {X 0,Y 431.177,Z 362.104,A -85,B 0,C 180,E1 -9289.026,E2 -9289.026} C_VEL
LIN {X 0,Y 431.14,Z 362.427,A -85,B 0,C 180,E1 -9290.018,E2 -9290.018} C_VEL
LIN {X 0,Y 431.174,Z 361.951,A -85,B 0,C 180,E1 -9291.708,E2 -9291.708} C_VEL
LIN {X 0,Y 431.266,Z 360.656,A -85,B 0,C 180,E1 -9293.024,E2 -9293.024} C_VEL
LIN {X 0,Y 431.427,Z 358.853,A -85,B 0,C 180,E1 -9294.183,E2 -9294.183} C_VEL
LIN {X 0,Y 431.634,Z 355.87,A -85,B 0,C 180,E1 -9295.562,E2 -9295.562} C_VEL
LIN {X 0,Y 431.903,Z 351.33,A -85,B 0,C 180,E1 -9297.105,E2 -9297.105} C_VEL
LIN {X 0,Y 432.27,Z 345.587,A -85,B 0,C 180,E1 -9298.604,E2 -9298.604} C_VEL
LIN {X 0,Y 432.772,Z 339.066,A -85,B 0,C 180,E1 -9299.958,E2 -9299.958} C_VEL
LIN {X 0,Y 433.324,Z 331.327,A -85,B 0,C 180,E1 -9301.266,E2 -9301.266} C_VEL
LIN {X 0,Y 434.068,Z 321.763,A -85,B 0,C 180,E1 -9302.562,E2 -9302.562} C_VEL
LIN {X 0,Y 434.653,Z 312.109,A -85,B 0,C 180,E1 -9303.628,E2 -9303.628} C_VEL
LIN {X 0,Y 435.399,Z 301.248,A -85,B 0,C 180,E1 -9304.592,E2 -9304.592} C_VEL
LIN {X 0,Y 436.049,Z 289.69,A -85,B 0,C 180,E1 -9305.394,E2 -9305.394} C_VEL
LIN {X 0,Y 436.53,Z 277.001,A -85,B 0,C 180,E1 -9306.061,E2 -9306.061} C_VEL
LIN {X 0,Y 436.956,Z 263.89,A -85,B 0,C 180,E1 -9306.538,E2 -9306.538} C_VEL
LIN {X 0,Y 437.161,Z 249.678,A -85,B 0,C 180,E1 -9306.842,E2 -9306.842} C_VEL
LIN {X 0,Y 438.127,Z 169.716,A -85,B 0,C 180,E1 -9308.186,E2 -9308.186} C_VEL
LIN {X 0,Y 434.262,Z 152.122,A -85,B 0,C 180,E1 -9308.715,E2 -9308.715} C_VEL
LIN {X 0,Y 433.92,Z 147.451,A -85,B 0,C 180,E1 -9309.774,E2 -9309.774} C_VEL
LIN {X 0,Y 432.335,Z 139.632,A -85,B 0,C 180,E1 -9311.662,E2 -9311.662} C_VEL
LIN {X 0,Y 432.333,Z 139.635,A -85,B 0,C 180,E1 -9314.348,E2 -9314.348} C_VEL
LIN {X 0,Y 432.302,Z 139.639,A -85,B 0,C 180,E1 -9317.019,E2 -9317.019} C_VEL
LIN {X 0,Y 432.289,Z 139.634,A -85,B 0,C 180,E1 -9319.828,E2 -9319.828} C_VEL
LIN {X 0,Y 432.304,Z 139.631,A -85,B 0,C 180,E1 -9323.022,E2 -9323.022} C_VEL
LIN {X 0,Y 432.333,Z 139.63,A -85,B 0,C 180,E1 -9326.002,E2 -9326.002} C_VEL
LIN {X 0,Y 432.338,Z 139.632,A -85,B 0,C 180,E1 -9329.492,E2 -9329.492} C_VEL
LIN {X 0,Y 432.318,Z 139.631,A -85,B 0,C 180,E1 -9331.872,E2 -9331.872} C_VEL
LIN {X 0,Y 432.346,Z 139.629,A -85,B 0,C 180,E1 -9335.548,E2 -9335.548} C_VEL
LIN {X 0,Y 432.322,Z 139.633,A -85,B 0,C 180,E1 -9339.045,E2 -9339.045} C_VEL
LIN {X 0,Y 432.315,Z 139.63,A -85,B 0,C 180,E1 -9342.009,E2 -9342.009} C_VEL
LIN {X 0,Y 432.325,Z 139.627,A -85,B 0,C 180,E1 -9344.924,E2 -9344.924} C_VEL
LIN {X 0,Y 432.448,Z 139.617,A -85,B 0,C 180,E1 -9347.803,E2 -9347.803} C_VEL
LIN {X 0,Y 432.446,Z 139.616,A -85,B 0,C 180,E1 -9351.59,E2 -9351.59} C_VEL
LIN {X 0,Y 432.551,Z 139.603,A -85,B 0,C 180,E1 -9354.406,E2 -9354.406} C_VEL
LIN {X 0,Y 432.596,Z 139.593,A -85,B 0,C 180,E1 -9358.138,E2 -9358.138} C_VEL
LIN {X 0,Y 432.621,Z 139.598,A -85,B 0,C 180,E1 -9360,E2 -9360} C_VEL
LIN {X 0,Y 432.558,Z 139.593,A -85,B 0,C 180,E1 -9362.794,E2 -9362.794} C_VEL
LIN {X 0,Y 432.571,Z 139.604,A -85,B 0,C 180,E1 -9365.594,E2 -9365.594} C_VEL
LIN {X 0,Y 432.45,Z 139.61,A -85,B 0,C 180,E1 -9368.411,E2 -9368.411} C_VEL
LIN {X 0,Y 432.461,Z 139.608,A -85,B 0,C 180,E1 -9372.197,E2 -9372.197} C_VEL
LIN {X 0,Y 432.427,Z 139.616,A -85,B 0,C 180,E1 -9376.039,E2 -9376.039} C_VEL
LIN {X 0,Y 432.389,Z 139.626,A -85,B 0,C 180,E1 -9379.485,E2 -9379.485} C_VEL
LIN {X 0,Y 432.319,Z 139.628,A -85,B 0,C 180,E1 -9382.964,E2 -9382.964} C_VEL
LIN {X 0,Y 432.339,Z 139.633,A -85,B 0,C 180,E1 -9385.002,E2 -9385.002} C_VEL
LIN {X 0,Y 432.341,Z 139.627,A -85,B 0,C 180,E1 -9388.126,E2 -9388.126} C_VEL
LIN {X 0,Y 432.322,Z 139.632,A -85,B 0,C 180,E1 -9391.346,E2 -9391.346} C_VEL
LIN {X 0,Y 432.34,Z 139.629,A -85,B 0,C 180,E1 -9394.677,E2 -9394.677} C_VEL
LIN {X 0,Y 432.334,Z 139.628,A -85,B 0,C 180,E1 -9398.151,E2 -9398.151} C_VEL
LIN {X 0,Y 432.322,Z 139.632,A -85,B 0,C 180,E1 -9401.799,E2 -9401.799} C_VEL
LIN {X 0,Y 432.336,Z 139.635,A -85,B 0,C 180,E1 -9404.347,E2 -9404.347} C_VEL
LIN {X 0,Y 432.319,Z 139.635,A -85,B 0,C 180,E1 -9407.016,E2 -9407.016} C_VEL
LIN {X 0,Y 432.334,Z 139.633,A -85,B 0,C 180,E1 -9409.821,E2 -9409.821} C_VEL
LIN {X 0,Y 432.307,Z 139.632,A -85,B 0,C 180,E1 -9413.022,E2 -9413.022} C_VEL
LIN {X 0,Y 432.362,Z 139.627,A -85,B 0,C 180,E1 -9415.997,E2 -9415.997} C_VEL
LIN {X 0,Y 432.35,Z 139.631,A -85,B 0,C 180,E1 -9419.49,E2 -9419.49} C_VEL
LIN {X 0,Y 432.465,Z 139.8,A -85,B 0,C 180,E1 -9422.08,E2 -9422.08} C_VEL
LIN {X 0,Y 435.137,Z 152.655,A -85,B 0,C 180,E1 -9424.752,E2 -9424.752} C_VEL
LIN {X 0,Y 435.504,Z 156.18,A -85,B 0,C 180,E1 -9425.446,E2 -9425.446} C_VEL
LIN {X 0,Y 434.402,Z 173.531,A -85,B 0,C 180,E1 -9428.653,E2 -9428.653} C_VEL
LIN {X 0,Y 433.633,Z 188.073,A -85,B 0,C 180,E1 -9431.307,E2 -9431.307} C_VEL
LIN {X 0,Y 437.197,Z 210.516,A -85,B 0,C 180,E1 -9431.887,E2 -9431.887} C_VEL
LIN {X 0,Y 437.621,Z 215.119,A -85,B 0,C 180,E1 -9431.987,E2 -9431.987} C_VEL
LIN {X 0,Y 436.741,Z 297.733,A -85,B 0,C 180,E1 -9433.403,E2 -9433.403} C_VEL
LIN {X 0,Y 436.123,Z 311.426,A -85,B 0,C 180,E1 -9433.83,E2 -9433.83} C_VEL
LIN {X 0,Y 435.504,Z 324.272,A -85,B 0,C 180,E1 -9434.437,E2 -9434.437} C_VEL
LIN {X 0,Y 434.731,Z 336.804,A -85,B 0,C 180,E1 -9435.249,E2 -9435.249} C_VEL
LIN {X 0,Y 434.007,Z 347.797,A -85,B 0,C 180,E1 -9436.162,E2 -9436.162} C_VEL
LIN {X 0,Y 433.314,Z 358.107,A -85,B 0,C 180,E1 -9437.233,E2 -9437.233} C_VEL
LIN {X 0,Y 432.692,Z 368.067,A -85,B 0,C 180,E1 -9438.523,E2 -9438.523} C_VEL
LIN {X 0,Y 432.06,Z 376.859,A -85,B 0,C 180,E1 -9439.929,E2 -9439.929} C_VEL
LIN {X 0,Y 431.699,Z 383.895,A -85,B 0,C 180,E1 -9441.339,E2 -9441.339} C_VEL
LIN {X 0,Y 431.414,Z 390.359,A -85,B 0,C 180,E1 -9442.982,E2 -9442.982} C_VEL
LIN {X 0,Y 431.259,Z 394.624,A -85,B 0,C 180,E1 -9444.389,E2 -9444.389} C_VEL
LIN {X 0,Y 431.268,Z 396.896,A -85,B 0,C 180,E1 -9445.326,E2 -9445.326} C_VEL
LIN {X 0,Y 431.198,Z 398.69,A -85,B 0,C 180,E1 -9446.262,E2 -9446.262} C_VEL
LIN {X 0,Y 431.283,Z 400.059,A -85,B 0,C 180,E1 -9447.198,E2 -9447.198} C_VEL
LIN {X 0,Y 431.224,Z 401.607,A -85,B 0,C 180,E1 -9449.066,E2 -9449.066} C_VEL
LIN {X 0,Y 431.229,Z 401.754,A -85,B 0,C 180,E1 -9450,E2 -9450} C_VEL
LIN {X 0,Y 431.242,Z 400.85,A -85,B 0,C 180,E1 -9451.868,E2 -9451.868} C_VEL
LIN {X 0,Y 431.284,Z 399.812,A -85,B 0,C 180,E1 -9452.802,E2 -9452.802} C_VEL
LIN {X 0,Y 431.202,Z 398.318,A -85,B 0,C 180,E1 -9453.738,E2 -9453.738} C_VEL
LIN {X 0,Y 431.282,Z 395.279,A -85,B 0,C 180,E1 -9455.142,E2 -9455.142} C_VEL
LIN {X 0,Y 431.291,Z 391.164,A -85,B 0,C 180,E1 -9456.55,E2 -9456.55} C_VEL
LIN {X 0,Y 431.569,Z 384.853,A -85,B 0,C 180,E1 -9458.192,E2 -9458.192} C_VEL
LIN {X 0,Y 431.853,Z 377.97,A -85,B 0,C 180,E1 -9459.602,E2 -9459.602} C_VEL
LIN {X 0,Y 432.345,Z 369.385,A -85,B 0,C 180,E1 -9461.011,E2 -9461.011} C_VEL
LIN {X 0,Y 432.868,Z 360.549,A -85,B 0,C 180,E1 -9462.185,E2 -9462.185} C_VEL
LIN {X 0,Y 433.395,Z 350.575,A -85,B 0,C 180,E1 -9463.269,E2 -9463.269} C_VEL
LIN {X 0,Y 434.072,Z 340.262,A -85,B 0,C 180,E1 -9464.175,E2 -9464.175} C_VEL
LIN {X 0,Y 434.705,Z 328.52,A -85,B 0,C 180,E1 -9464.991,E2 -9464.991} C_VEL
LIN {X 0,Y 435.257,Z 316.311,A -85,B 0,C 180,E1 -9465.631,E2 -9465.631} C_VEL
LIN {X 0,Y 435.815,Z 303.027,A -85,B 0,C 180,E1 -9466.121,E2 -9466.121} C_VEL
LIN {X 0,Y 436.104,Z 289.973,A -85,B 0,C 180,E1 -9466.411,E2 -9466.411} C_VEL
LIN {X 0,Y 436.643,Z 212.665,A -85,B 0,C 180,E1 -9467.701,E2 -9467.701} C_VEL
LIN {X 0,Y 433.276,Z 188.668,A -85,B 0,C 180,E1 -9468.253,E2 -9468.253} C_VEL
LIN {X 0,Y 434.123,Z 171.376,A -85,B 0,C 180,E1 -9471.361,E2 -9471.361} C_VEL
LIN {X 0,Y 435.038,Z 155.046,A -85,B 0,C 180,E1 -9474.327,E2 -9474.327} C_VEL
LIN {X 0,Y 434.636,Z 150.947,A -85,B 0,C 180,E1 -9475.107,E2 -9475.107} C_VEL
LIN {X 0,Y 432.419,Z 139.623,A -85,B 0,C 180,E1 -9477.397,E2 -9477.397} C_VEL
LIN {X 0,Y 432.349,Z 139.631,A -85,B 0,C 180,E1 -9480.51,E2 -9480.51} C_VEL
LIN {X 0,Y 432.361,Z 139.631,A -85,B 0,C 180,E1 -9484.003,E2 -9484.003} C_VEL
LIN {X 0,Y 432.324,Z 139.629,A -85,B 0,C 180,E1 -9487.197,E2 -9487.197} C_VEL
LIN {X 0,Y 432.342,Z 139.63,A -85,B 0,C 180,E1 -9490.18,E2 -9490.18} C_VEL
LIN {X 0,Y 432.318,Z 139.63,A -85,B 0,C 180,E1 -9493.061,E2 -9493.061} C_VEL
LIN {X 0,Y 432.334,Z 139.635,A -85,B 0,C 180,E1 -9495.664,E2 -9495.664} C_VEL
LIN {X 0,Y 432.333,Z 139.628,A -85,B 0,C 180,E1 -9498.398,E2 -9498.398} C_VEL
LIN {X 0,Y 432.335,Z 139.631,A -85,B 0,C 180,E1 -9501.85,E2 -9501.85} C_VEL
LIN {X 0,Y 432.338,Z 139.633,A -85,B 0,C 180,E1 -9505.322,E2 -9505.322} C_VEL
LIN {X 0,Y 432.321,Z 139.63,A -85,B 0,C 180,E1 -9508.654,E2 -9508.654} C_VEL
LIN {X 0,Y 432.382,Z 139.623,A -85,B 0,C 180,E1 -9511.876,E2 -9511.876} C_VEL
LIN {X 0,Y 432.349,Z 139.63,A -85,B 0,C 180,E1 -9514.998,E2 -9514.998} C_VEL
LIN {X 0,Y 432.358,Z 139.625,A -85,B 0,C 180,E1 -9518.046,E2 -9518.046} C_VEL
LIN {X 0,Y 432.384,Z 139.628,A -85,B 0,C 180,E1 -9521.029,E2 -9521.029} C_VEL
LIN {X 0,Y 432.43,Z 139.615,A -85,B 0,C 180,E1 -9523.961,E2 -9523.961} C_VEL
LIN {X 0,Y 432.459,Z 139.612,A -85,B 0,C 180,E1 -9527.803,E2 -9527.803} C_VEL
LIN {X 0,Y 432.463,Z 139.612,A -85,B 0,C 180,E1 -9531.59,E2 -9531.59} C_VEL
LIN {X 0,Y 432.586,Z 139.599,A -85,B 0,C 180,E1 -9534.406,E2 -9534.406} C_VEL
LIN {X 0,Y 432.605,Z 139.595,A -85,B 0,C 180,E1 -9538.138,E2 -9538.138} C_VEL
LIN {X 0,Y 432.732,Z 139.579,A -85,B 0,C 180,E1 -9540,E2 -9540} C_VEL
LIN {X 0,Y 432.603,Z 139.599,A -85,B 0,C 180,E1 -9542.793,E2 -9542.793} C_VEL
LIN {X 0,Y 432.564,Z 139.606,A -85,B 0,C 180,E1 -9546.53,E2 -9546.53} C_VEL
LIN {X 0,Y 432.441,Z 139.614,A -85,B 0,C 180,E1 -9549.353,E2 -9549.353} C_VEL
LIN {X 0,Y 432.43,Z 139.618,A -85,B 0,C 180,E1 -9552.803,E2 -9552.803} C_VEL
LIN {X 0,Y 432.411,Z 139.623,A -85,B 0,C 180,E1 -9556.478,E2 -9556.478} C_VEL
LIN {X 0,Y 432.338,Z 139.631,A -85,B 0,C 180,E1 -9559.96,E2 -9559.96} C_VEL
LIN {X 0,Y 432.317,Z 139.63,A -85,B 0,C 180,E1 -9562.964,E2 -9562.964} C_VEL
LIN {X 0,Y 432.36,Z 139.631,A -85,B 0,C 180,E1 -9566.033,E2 -9566.033} C_VEL
LIN {X 0,Y 432.341,Z 139.627,A -85,B 0,C 180,E1 -9569.187,E2 -9569.187} C_VEL
LIN {X 0,Y 432.322,Z 139.631,A -85,B 0,C 180,E1 -9572.443,E2 -9572.443} C_VEL
LIN {X 0,Y 432.343,Z 139.631,A -85,B 0,C 180,E1 -9575.632,E2 -9575.632} C_VEL
LIN {X 0,Y 432.354,Z 139.627,A -85,B 0,C 180,E1 -9579.342,E2 -9579.342} C_VEL
LIN {X 0,Y 432.333,Z 139.634,A -85,B 0,C 180,E1 -9581.797,E2 -9581.797} C_VEL
LIN {X 0,Y 432.332,Z 139.628,A -85,B 0,C 180,E1 -9584.347,E2 -9584.347} C_VEL
LIN {X 0,Y 432.319,Z 139.631,A -85,B 0,C 180,E1 -9587.016,E2 -9587.016} C_VEL
LIN {X 0,Y 432.332,Z 139.632,A -85,B 0,C 180,E1 -9589.821,E2 -9589.821} C_VEL
LIN {X 0,Y 432.305,Z 139.633,A -85,B 0,C 180,E1 -9593.022,E2 -9593.022} C_VEL
LIN {X 0,Y 432.356,Z 139.626,A -85,B 0,C 180,E1 -9595.997,E2 -9595.997} C_VEL
LIN {X 0,Y 432.346,Z 139.631,A -85,B 0,C 180,E1 -9599.49,E2 -9599.49} C_VEL
LIN {X 0,Y 432.39,Z 139.624,A -85,B 0,C 180,E1 -9602.928,E2 -9602.928} C_VEL
LIN {X 0,Y 432.369,Z 139.623,A -85,B 0,C 180,E1 -9606.023,E2 -9606.023} C_VEL
LIN {X 0,Y 432.35,Z 139.632,A -85,B 0,C 180,E1 -9609.046,E2 -9609.046} C_VEL
LIN {X 0,Y 432.36,Z 139.624,A -85,B 0,C 180,E1 -9612.011,E2 -9612.011} C_VEL
LIN {X 0,Y 432.395,Z 139.627,A -85,B 0,C 180,E1 -9614.927,E2 -9614.927} C_VEL
LIN {X 0,Y 432.459,Z 139.612,A -85,B 0,C 180,E1 -9617.804,E2 -9617.804} C_VEL
LIN {X 0,Y 432.464,Z 139.612,A -85,B 0,C 180,E1 -9621.59,E2 -9621.59} C_VEL
LIN {X 0,Y 432.587,Z 139.599,A -85,B 0,C 180,E1 -9624.406,E2 -9624.406} C_VEL
LIN {X 0,Y 432.605,Z 139.6,A -85,B 0,C 180,E1 -9628.138,E2 -9628.138} C_VEL
LIN {X 0,Y 432.582,Z 139.675,A -85,B 0,C 180,E1 -9629.127,E2 -9629.127} C_VEL
LIN {X 0,Y 433.732,Z 146.49,A -85,B 0,C 180,E1 -9630.696,E2 -9630.696} C_VEL
LIN {X 0,Y 433.7,Z 151.548,A -85,B 0,C 180,E1 -9631.81,E2 -9631.81} C_VEL
LIN {X 0,Y 433.263,Z 152.778,A -85,B 0,C 180,E1 -9631.856,E2 -9631.856} C_VEL
LIN {X 0,Y 428.7,Z 162.365,A -85,B 0,C 180,E1 -9631.842,E2 -9631.842} C_VEL
LIN {X 0,Y 427.78,Z 166.523,A -85,B 0,C 180,E1 -9631.856,E2 -9631.856} C_VEL
LIN {X 0,Y 427.939,Z 169.861,A -85,B 0,C 180,E1 -9631.887,E2 -9631.887} C_VEL
LIN {X 0,Y 430.156,Z 180.785,A -85,B 0,C 180,E1 -9632.214,E2 -9632.214} C_VEL
LIN {X 0,Y 430.249,Z 183.038,A -85,B 0,C 180,E1 -9632.262,E2 -9632.262} C_VEL
LIN {X 0,Y 429.274,Z 259.738,A -85,B 0,C 180,E1 -9633.578,E2 -9633.578} C_VEL
LIN {X 0,Y 428.943,Z 272.782,A -85,B 0,C 180,E1 -9633.993,E2 -9633.993} C_VEL
LIN {X 0,Y 428.562,Z 285.334,A -85,B 0,C 180,E1 -9634.586,E2 -9634.586} C_VEL
LIN {X 0,Y 428.041,Z 296.577,A -85,B 0,C 180,E1 -9635.299,E2 -9635.299} C_VEL
LIN {X 0,Y 427.469,Z 308.199,A -85,B 0,C 180,E1 -9636.253,E2 -9636.253} C_VEL
LIN {X 0,Y 426.797,Z 318.711,A -85,B 0,C 180,E1 -9637.332,E2 -9637.332} C_VEL
LIN {X 0,Y 426.129,Z 328.157,A -85,B 0,C 180,E1 -9638.536,E2 -9638.536} C_VEL
LIN {X 0,Y 425.529,Z 337.272,A -85,B 0,C 180,E1 -9639.987,E2 -9639.987} C_VEL
LIN {X 0,Y 425.089,Z 344.608,A -85,B 0,C 180,E1 -9641.443,E2 -9641.443} C_VEL
LIN {X 0,Y 424.768,Z 350.278,A -85,B 0,C 180,E1 -9642.858,E2 -9642.858} C_VEL
LIN {X 0,Y 424.486,Z 355.033,A -85,B 0,C 180,E1 -9644.38,E2 -9644.38} C_VEL
LIN {X 0,Y 424.26,Z 358.945,A -85,B 0,C 180,E1 -9646.099,E2 -9646.099} C_VEL
LIN {X 0,Y 424.112,Z 360.922,A -85,B 0,C 180,E1 -9647.354,E2 -9647.354} C_VEL
LIN {X 0,Y 424.074,Z 362.489,A -85,B 0,C 180,E1 -9649.155,E2 -9649.155} C_VEL
LIN {X 0,Y 424.06,Z 362.76,A -85,B 0,C 180,E1 -9650.367,E2 -9650.367} C_VEL
LIN {X 0,Y 424.116,Z 362.187,A -85,B 0,C 180,E1 -9651.879,E2 -9651.879} C_VEL
LIN {X 0,Y 424.222,Z 360.553,A -85,B 0,C 180,E1 -9653.429,E2 -9653.429} C_VEL
LIN {X 0,Y 424.46,Z 357.826,A -85,B 0,C 180,E1 -9654.975,E2 -9654.975} C_VEL
LIN {X 0,Y 424.742,Z 353.462,A -85,B 0,C 180,E1 -9656.682,E2 -9656.682} C_VEL
LIN {X 0,Y 425.157,Z 347.586,A -85,B 0,C 180,E1 -9658.376,E2 -9658.376} C_VEL
LIN {X 0,Y 425.728,Z 340.382,A -85,B 0,C 180,E1 -9659.959,E2 -9659.959} C_VEL
LIN {X 0,Y 426.337,Z 332.557,A -85,B 0,C 180,E1 -9661.335,E2 -9661.335} C_VEL
LIN {X 0,Y 427.049,Z 323.582,A -85,B 0,C 180,E1 -9662.614,E2 -9662.614} C_VEL
LIN {X 0,Y 427.771,Z 313.195,A -85,B 0,C 180,E1 -9663.803,E2 -9663.803} C_VEL
LIN {X 0,Y 428.575,Z 302.009,A -85,B 0,C 180,E1 -9664.826,E2 -9664.826} C_VEL
LIN {X 0,Y 429.31,Z 290.027,A -85,B 0,C 180,E1 -9665.676,E2 -9665.676} C_VEL
LIN {X 0,Y 429.805,Z 277.34,A -85,B 0,C 180,E1 -9666.355,E2 -9666.355} C_VEL
LIN {X 0,Y 430.243,Z 264.332,A -85,B 0,C 180,E1 -9666.838,E2 -9666.838} C_VEL
LIN {X 0,Y 430.49,Z 249.362,A -85,B 0,C 180,E1 -9667.16,E2 -9667.16} C_VEL
LIN {X 0,Y 431.439,Z 170.292,A -85,B 0,C 180,E1 -9668.516,E2 -9668.516} C_VEL
LIN {X 0,Y 427.384,Z 152.521,A -85,B 0,C 180,E1 -9669.056,E2 -9669.056} C_VEL
LIN {X 0,Y 426.681,Z 147.128,A -85,B 0,C 180,E1 -9670.318,E2 -9670.318} C_VEL
LIN {X 0,Y 425.278,Z 140.511,A -85,B 0,C 180,E1 -9671.957,E2 -9671.957} C_VEL
LIN {X 0,Y 425.284,Z 140.512,A -85,B 0,C 180,E1 -9675.283,E2 -9675.283} C_VEL
LIN {X 0,Y 425.247,Z 140.518,A -85,B 0,C 180,E1 -9678.618,E2 -9678.618} C_VEL
LIN {X 0,Y 425.28,Z 140.511,A -85,B 0,C 180,E1 -9681.1,E2 -9681.1} C_VEL
LIN {X 0,Y 425.295,Z 140.506,A -85,B 0,C 180,E1 -9684.664,E2 -9684.664} C_VEL
LIN {X 0,Y 425.253,Z 140.513,A -85,B 0,C 180,E1 -9688.072,E2 -9688.072} C_VEL
LIN {X 0,Y 425.295,Z 140.507,A -85,B 0,C 180,E1 -9691.365,E2 -9691.365} C_VEL
LIN {X 0,Y 425.251,Z 140.514,A -85,B 0,C 180,E1 -9694.552,E2 -9694.552} C_VEL
LIN {X 0,Y 425.289,Z 140.502,A -85,B 0,C 180,E1 -9697.731,E2 -9697.731} C_VEL
LIN {X 0,Y 425.319,Z 140.502,A -85,B 0,C 180,E1 -9700.702,E2 -9700.702} C_VEL
LIN {X 0,Y 425.309,Z 140.505,A -85,B 0,C 180,E1 -9703.685,E2 -9703.685} C_VEL
LIN {X 0,Y 425.401,Z 140.493,A -85,B 0,C 180,E1 -9707.598,E2 -9707.598} C_VEL
LIN {X 0,Y 425.394,Z 140.493,A -85,B 0,C 180,E1 -9711.449,E2 -9711.449} C_VEL
LIN {X 0,Y 425.509,Z 140.48,A -85,B 0,C 180,E1 -9714.313,E2 -9714.313} C_VEL
LIN {X 0,Y 425.565,Z 140.469,A -85,B 0,C 180,E1 -9718.107,E2 -9718.107} C_VEL
LIN {X 0,Y 425.573,Z 140.475,A -85,B 0,C 180,E1 -9720,E2 -9720} C_VEL
LIN {X 0,Y 425.513,Z 140.47,A -85,B 0,C 180,E1 -9722.84,E2 -9722.84} C_VEL
LIN {X 0,Y 425.526,Z 140.482,A -85,B 0,C 180,E1 -9725.687,E2 -9725.687} C_VEL
LIN {X 0,Y 425.398,Z 140.488,A -85,B 0,C 180,E1 -9728.551,E2 -9728.551} C_VEL
LIN {X 0,Y 425.414,Z 140.485,A -85,B 0,C 180,E1 -9732.402,E2 -9732.402} C_VEL
LIN {X 0,Y 425.387,Z 140.492,A -85,B 0,C 180,E1 -9736.312,E2 -9736.312} C_VEL
LIN {X 0,Y 425.33,Z 140.503,A -85,B 0,C 180,E1 -9739.635,E2 -9739.635} C_VEL
LIN {X 0,Y 425.306,Z 140.507,A -85,B 0,C 180,E1 -9743.365,E2 -9743.365} C_VEL
LIN {X 0,Y 425.299,Z 140.502,A -85,B 0,C 180,E1 -9746.499,E2 -9746.499} C_VEL
LIN {X 0,Y 425.285,Z 140.504,A -85,B 0,C 180,E1 -9749.72,E2 -9749.72} C_VEL
LIN {X 0,Y 425.284,Z 140.509,A -85,B 0,C 180,E1 -9753.048,E2 -9753.048} C_VEL
LIN {X 0,Y 425.284,Z 140.508,A -85,B 0,C 180,E1 -9755.929,E2 -9755.929} C_VEL
LIN {X 0,Y 425.267,Z 140.513,A -85,B 0,C 180,E1 -9759.038,E2 -9759.038} C_VEL
LIN {X 0,Y 425.271,Z 140.513,A -85,B 0,C 180,E1 -9762.654,E2 -9762.654} C_VEL
LIN {X 0,Y 425.263,Z 140.513,A -85,B 0,C 180,E1 -9766.044,E2 -9766.044} C_VEL
LIN {X 0,Y 425.279,Z 140.511,A -85,B 0,C 180,E1 -9769.48,E2 -9769.48} C_VEL
LIN {X 0,Y 425.278,Z 140.506,A -85,B 0,C 180,E1 -9772.489,E2 -9772.489} C_VEL
LIN {X 0,Y 425.31,Z 140.504,A -85,B 0,C 180,E1 -9775.817,E2 -9775.817} C_VEL
LIN {X 0,Y 425.293,Z 140.511,A -85,B 0,C 180,E1 -9779.239,E2 -9779.239} C_VEL
LIN {X 0,Y 425.379,Z 140.599,A -85,B 0,C 180,E1 -9781.741,E2 -9781.741} C_VEL
LIN {X 0,Y 427.835,Z 151.971,A -85,B 0,C 180,E1 -9784.176,E2 -9784.176} C_VEL
LIN {X 0,Y 428.639,Z 157.415,A -85,B 0,C 180,E1 -9785.285,E2 -9785.285} C_VEL
LIN {X 0,Y 427.368,Z 176.096,A -85,B 0,C 180,E1 -9788.79,E2 -9788.79} C_VEL
LIN {X 0,Y 426.748,Z 187.753,A -85,B 0,C 180,E1 -9790.953,E2 -9790.953} C_VEL
LIN {X 0,Y 430.449,Z 210.517,A -85,B 0,C 180,E1 -9791.557,E2 -9791.557} C_VEL
LIN {X 0,Y 430.937,Z 216.9,A -85,B 0,C 180,E1 -9791.695,E2 -9791.695} C_VEL
LIN {X 0,Y 430.005,Z 297.487,A -85,B 0,C 180,E1 -9793.105,E2 -9793.105} C_VEL
LIN {X 0,Y 429.374,Z 311.122,A -85,B 0,C 180,E1 -9793.538,E2 -9793.538} C_VEL
LIN {X 0,Y 428.743,Z 323.424,A -85,B 0,C 180,E1 -9794.125,E2 -9794.125} C_VEL
LIN {X 0,Y 427.994,Z 335.276,A -85,B 0,C 180,E1 -9794.889,E2 -9794.889} C_VEL
LIN {X 0,Y 427.203,Z 346.509,A -85,B 0,C 180,E1 -9795.818,E2 -9795.818} C_VEL
LIN {X 0,Y 426.392,Z 357.011,A -85,B 0,C 180,E1 -9796.901,E2 -9796.901} C_VEL
LIN {X 0,Y 425.846,Z 366.299,A -85,B 0,C 180,E1 -9798.094,E2 -9798.094} C_VEL
LIN {X 0,Y 425.068,Z 375.332,A -85,B 0,C 180,E1 -9799.521,E2 -9799.521} C_VEL
LIN {X 0,Y 424.671,Z 382.63,A -85,B 0,C 180,E1 -9800.954,E2 -9800.954} C_VEL
LIN {X 0,Y 424.376,Z 388.484,A -85,B 0,C 180,E1 -9802.387,E2 -9802.387} C_VEL
LIN {X 0,Y 424.21,Z 392.881,A -85,B 0,C 180,E1 -9803.741,E2 -9803.741} C_VEL
LIN {X 0,Y 424.196,Z 396.634,A -85,B 0,C 180,E1 -9805.248,E2 -9805.248} C_VEL
LIN {X 0,Y 424.108,Z 398.408,A -85,B 0,C 180,E1 -9806.199,E2 -9806.199} C_VEL
LIN {X 0,Y 424.178,Z 399.767,A -85,B 0,C 180,E1 -9807.151,E2 -9807.151} C_VEL
LIN {X 0,Y 424.167,Z 400.728,A -85,B 0,C 180,E1 -9808.101,E2 -9808.101} C_VEL
LIN {X 0,Y 424.141,Z 401.294,A -85,B 0,C 180,E1 -9809.05,E2 -9809.05} C_VEL
LIN {X 0,Y 424.142,Z 401.425,A -85,B 0,C 180,E1 -9810,E2 -9810} C_VEL
LIN {X 0,Y 424.167,Z 400.501,A -85,B 0,C 180,E1 -9811.899,E2 -9811.899} C_VEL
LIN {X 0,Y 424.195,Z 399.45,A -85,B 0,C 180,E1 -9812.849,E2 -9812.849} C_VEL
LIN {X 0,Y 424.112,Z 397.935,A -85,B 0,C 180,E1 -9813.8,E2 -9813.8} C_VEL
LIN {X 0,Y 424.191,Z 394.873,A -85,B 0,C 180,E1 -9815.228,E2 -9815.228} C_VEL
LIN {X 0,Y 424.224,Z 390.734,A -85,B 0,C 180,E1 -9816.659,E2 -9816.659} C_VEL
LIN {X 0,Y 424.5,Z 384.395,A -85,B 0,C 180,E1 -9818.329,E2 -9818.329} C_VEL
LIN {X 0,Y 424.827,Z 377.482,A -85,B 0,C 180,E1 -9819.763,E2 -9819.763} C_VEL
LIN {X 0,Y 425.221,Z 370.422,A -85,B 0,C 180,E1 -9820.957,E2 -9820.957} C_VEL
LIN {X 0,Y 425.796,Z 361.92,A -85,B 0,C 180,E1 -9822.148,E2 -9822.148} C_VEL
LIN {X 0,Y 426.352,Z 351.392,A -85,B 0,C 180,E1 -9823.343,E2 -9823.343} C_VEL
LIN {X 0,Y 427.06,Z 340.988,A -85,B 0,C 180,E1 -9824.291,E2 -9824.291} C_VEL
LIN {X 0,Y 427.695,Z 329.579,A -85,B 0,C 180,E1 -9825.121,E2 -9825.121} C_VEL
LIN {X 0,Y 428.254,Z 317.891,A -85,B 0,C 180,E1 -9825.771,E2 -9825.771} C_VEL
LIN {X 0,Y 428.866,Z 304.459,A -85,B 0,C 180,E1 -9826.298,E2 -9826.298} C_VEL
LIN {X 0,Y 429.213,Z 291.263,A -85,B 0,C 180,E1 -9826.621,E2 -9826.621} C_VEL
LIN {X 0,Y 429.925,Z 214.276,A -85,B 0,C 180,E1 -9827.922,E2 -9827.922} C_VEL
LIN {X 0,Y 426.313,Z 188.288,A -85,B 0,C 180,E1 -9828.533,E2 -9828.533} C_VEL
LIN {X 0,Y 427.288,Z 169.475,A -85,B 0,C 180,E1 -9831.974,E2 -9831.974} C_VEL
LIN {X 0,Y 428.073,Z 155.873,A -85,B 0,C 180,E1 -9834.491,E2 -9834.491} C_VEL
LIN {X 0,Y 427.329,Z 150.331,A -85,B 0,C 180,E1 -9835.576,E2 -9835.576} C_VEL
LIN {X 0,Y 425.387,Z 140.501,A -85,B 0,C 180,E1 -9837.588,E2 -9837.588} C_VEL
LIN {X 0,Y 425.289,Z 140.509,A -85,B 0,C 180,E1 -9840.816,E2 -9840.816} C_VEL
LIN {X 0,Y 425.313,Z 140.505,A -85,B 0,C 180,E1 -9844.288,E2 -9844.288} C_VEL
LIN {X 0,Y 425.281,Z 140.511,A -85,B 0,C 180,E1 -9847.694,E2 -9847.694} C_VEL
LIN {X 0,Y 425.285,Z 140.506,A -85,B 0,C 180,E1 -9850.521,E2 -9850.521} C_VEL
LIN {X 0,Y 425.258,Z 140.512,A -85,B 0,C 180,E1 -9853.351,E2 -9853.351} C_VEL
LIN {X 0,Y 425.258,Z 140.509,A -85,B 0,C 180,E1 -9856.649,E2 -9856.649} C_VEL
LIN {X 0,Y 425.286,Z 140.509,A -85,B 0,C 180,E1 -9859.872,E2 -9859.872} C_VEL
LIN {X 0,Y 425.278,Z 140.506,A -85,B 0,C 180,E1 -9862.488,E2 -9862.488} C_VEL
LIN {X 0,Y 425.306,Z 140.506,A -85,B 0,C 180,E1 -9865.817,E2 -9865.817} C_VEL
LIN {X 0,Y 425.291,Z 140.51,A -85,B 0,C 180,E1 -9869.239,E2 -9869.239} C_VEL
LIN {X 0,Y 425.349,Z 140.498,A -85,B 0,C 180,E1 -9872.442,E2 -9872.442} C_VEL
LIN {X 0,Y 425.35,Z 140.501,A -85,B 0,C 180,E1 -9875.602,E2 -9875.602} C_VEL
LIN {X 0,Y 425.293,Z 140.506,A -85,B 0,C 180,E1 -9878.681,E2 -9878.681} C_VEL
LIN {X 0,Y 425.322,Z 140.502,A -85,B 0,C 180,E1 -9881.702,E2 -9881.702} C_VEL
LIN {X 0,Y 425.348,Z 140.501,A -85,B 0,C 180,E1 -9884.67,E2 -9884.67} C_VEL
LIN {X 0,Y 425.412,Z 140.491,A -85,B 0,C 180,E1 -9887.598,E2 -9887.598} C_VEL
LIN {X 0,Y 425.408,Z 140.492,A -85,B 0,C 180,E1 -9891.449,E2 -9891.449} C_VEL
LIN {X 0,Y 425.542,Z 140.475,A -85,B 0,C 180,E1 -9894.313,E2 -9894.313} C_VEL
LIN {X 0,Y 425.574,Z 140.471,A -85,B 0,C 180,E1 -9898.107,E2 -9898.107} C_VEL
LIN {X 0,Y 425.701,Z 140.454,A -85,B 0,C 180,E1 -9900,E2 -9900} C_VEL
LIN {X 0,Y 425.555,Z 140.477,A -85,B 0,C 180,E1 -9902.84,E2 -9902.84} C_VEL
LIN {X 0,Y 425.523,Z 140.482,A -85,B 0,C 180,E1 -9906.639,E2 -9906.639} C_VEL
LIN {X 0,Y 425.4,Z 140.491,A -85,B 0,C 180,E1 -9909.509,E2 -9909.509} C_VEL
LIN {X 0,Y 425.393,Z 140.494,A -85,B 0,C 180,E1 -9912.904,E2 -9912.904} C_VEL
LIN {X 0,Y 425.36,Z 140.5,A -85,B 0,C 180,E1 -9916.605,E2 -9916.605} C_VEL
LIN {X 0,Y 425.327,Z 140.501,A -85,B 0,C 180,E1 -9919.635,E2 -9919.635} C_VEL
LIN {X 0,Y 425.287,Z 140.511,A -85,B 0,C 180,E1 -9922.339,E2 -9922.339} C_VEL
LIN {X 0,Y 425.29,Z 140.506,A -85,B 0,C 180,E1 -9925.446,E2 -9925.446} C_VEL
LIN {X 0,Y 425.347,Z 140.5,A -85,B 0,C 180,E1 -9927.558,E2 -9927.558} C_VEL
LIN {X 0,Y 425.287,Z 140.506,A -85,B 0,C 180,E1 -9930.816,E2 -9930.816} C_VEL
LIN {X 0,Y 425.31,Z 140.505,A -85,B 0,C 180,E1 -9934.288,E2 -9934.288} C_VEL
LIN {X 0,Y 425.279,Z 140.512,A -85,B 0,C 180,E1 -9937.694,E2 -9937.694} C_VEL
LIN {X 0,Y 425.283,Z 140.506,A -85,B 0,C 180,E1 -9940.521,E2 -9940.521} C_VEL
LIN {X 0,Y 425.256,Z 140.512,A -85,B 0,C 180,E1 -9943.351,E2 -9943.351} C_VEL
LIN {X 0,Y 425.256,Z 140.509,A -85,B 0,C 180,E1 -9946.649,E2 -9946.649} C_VEL
LIN {X 0,Y 425.284,Z 140.509,A -85,B 0,C 180,E1 -9949.873,E2 -9949.873} C_VEL
LIN {X 0,Y 425.276,Z 140.507,A -85,B 0,C 180,E1 -9952.489,E2 -9952.489} C_VEL
LIN {X 0,Y 425.304,Z 140.506,A -85,B 0,C 180,E1 -9955.817,E2 -9955.817} C_VEL
LIN {X 0,Y 425.289,Z 140.511,A -85,B 0,C 180,E1 -9959.239,E2 -9959.239} C_VEL
LIN {X 0,Y 425.348,Z 140.498,A -85,B 0,C 180,E1 -9962.442,E2 -9962.442} C_VEL
LIN {X 0,Y 425.349,Z 140.5,A -85,B 0,C 180,E1 -9965.602,E2 -9965.602} C_VEL
LIN {X 0,Y 425.293,Z 140.507,A -85,B 0,C 180,E1 -9968.682,E2 -9968.682} C_VEL
LIN {X 0,Y 425.321,Z 140.502,A -85,B 0,C 180,E1 -9971.702,E2 -9971.702} C_VEL
LIN {X 0,Y 425.348,Z 140.501,A -85,B 0,C 180,E1 -9974.671,E2 -9974.671} C_VEL
LIN {X 0,Y 425.412,Z 140.49,A -85,B 0,C 180,E1 -9977.598,E2 -9977.598} C_VEL
LIN {X 0,Y 425.408,Z 140.491,A -85,B 0,C 180,E1 -9981.449,E2 -9981.449} C_VEL
LIN {X 0,Y 425.542,Z 140.476,A -85,B 0,C 180,E1 -9984.313,E2 -9984.313} C_VEL
LIN {X 0,Y 425.574,Z 140.475,A -85,B 0,C 180,E1 -9988.107,E2 -9988.107} C_VEL
LIN {X 0,Y 425.54,Z 140.609,A -85,B 0,C 180,E1 -9988.965,E2 -9988.965} C_VEL
LIN {X 0,Y 426.801,Z 148.11,A -85,B 0,C 180,E1 -9990.708,E2 -9990.708} C_VEL
LIN {X 0,Y 426.775,Z 152.005,A -85,B 0,C 180,E1 -9991.569,E2 -9991.569} C_VEL
LIN {X 0,Y 430.293,Z 169.926,A -85,B 0,C 180,E1 -9992.036,E2 -9992.036} C_VEL
LIN {X 0,Y 430.249,Z 183.038,A -85,B 0,C 180,E1 -9992.262,E2 -9992.262} C_VEL
LIN {X 0,Y 429.474,Z 188.881,A -85,B 0,C 180,E1 -9992.332,E2 -9992.332} C_VEL
LIN {X 0,Y 423.687,Z 207.847,A -85,B 0,C 180,E1 -9992.443,E2 -9992.443} C_VEL
LIN {X 0,Y 423.009,Z 213.686,A -85,B 0,C 180,E1 -9992.52,E2 -9992.52} C_VEL
LIN {X 0,Y 422.4,Z 260.418,A -85,B 0,C 180,E1 -9993.349,E2 -9993.349} C_VEL
LIN {X 0,Y 422.06,Z 273.366,A -85,B 0,C 180,E1 -9993.772,E2 -9993.772} C_VEL
LIN {X 0,Y 421.669,Z 285.632,A -85,B 0,C 180,E1 -9994.361,E2 -9994.361} C_VEL
LIN {X 0,Y 421.109,Z 297.675,A -85,B 0,C 180,E1 -9995.147,E2 -9995.147} C_VEL
LIN {X 0,Y 420.506,Z 309.174,A -85,B 0,C 180,E1 -9996.116,E2 -9996.116} C_VEL
LIN {X 0,Y 419.809,Z 319.573,A -85,B 0,C 180,E1 -9997.213,E2 -9997.213} C_VEL
LIN {X 0,Y 419.137,Z 328.583,A -85,B 0,C 180,E1 -9998.391,E2 -9998.391} C_VEL
LIN {X 0,Y 418.611,Z 336.56,A -85,B 0,C 180,E1 -9999.665,E2 -9999.665} C_VEL
LIN {X 0,Y 418.106,Z 344.083,A -85,B 0,C 180,E1 -10001.146,E2 -10001.146} C_VEL
LIN {X 0,Y 417.737,Z 350.113,A -85,B 0,C 180,E1 -10002.634,E2 -10002.634} C_VEL
LIN {X 0,Y 417.461,Z 354.862,A -85,B 0,C 180,E1 -10004.129,E2 -10004.129} C_VEL
LIN {X 0,Y 417.213,Z 358.472,A -85,B 0,C 180,E1 -10005.636,E2 -10005.636} C_VEL
LIN {X 0,Y 417.11,Z 360.259,A -85,B 0,C 180,E1 -10006.645,E2 -10006.645} C_VEL
LIN {X 0,Y 417.019,Z 361.618,A -85,B 0,C 180,E1 -10007.659,E2 -10007.659} C_VEL
LIN {X 0,Y 417.008,Z 362.879,A -85,B 0,C 180,E1 -10009.302,E2 -10009.302} C_VEL
LIN {X 0,Y 416.959,Z 363.038,A -85,B 0,C 180,E1 -10010.73,E2 -10010.73} C_VEL
LIN {X 0,Y 417.033,Z 362.429,A -85,B 0,C 180,E1 -10012.047,E2 -10012.047} C_VEL
LIN {X 0,Y 417.204,Z 360.392,A -85,B 0,C 180,E1 -10013.847,E2 -10013.847} C_VEL
LIN {X 0,Y 417.474,Z 357.431,A -85,B 0,C 180,E1 -10015.422,E2 -10015.422} C_VEL
LIN {X 0,Y 417.762,Z 353.241,A -85,B 0,C 180,E1 -10017.015,E2 -10017.015} C_VEL
LIN {X 0,Y 418.176,Z 347.706,A -85,B 0,C 180,E1 -10018.6,E2 -10018.6} C_VEL
LIN {X 0,Y 418.788,Z 340.375,A -85,B 0,C 180,E1 -10020.229,E2 -10020.229} C_VEL
LIN {X 0,Y 419.439,Z 332.808,A -85,B 0,C 180,E1 -10021.575,E2 -10021.575} C_VEL
LIN {X 0,Y 420.235,Z 323.477,A -85,B 0,C 180,E1 -10022.918,E2 -10022.918} C_VEL
LIN {X 0,Y 421.028,Z 312.819,A -85,B 0,C 180,E1 -10024.145,E2 -10024.145} C_VEL
LIN {X 0,Y 421.874,Z 301.404,A -85,B 0,C 180,E1 -10025.187,E2 -10025.187} C_VEL
LIN {X 0,Y 422.617,Z 289.361,A -85,B 0,C 180,E1 -10026.035,E2 -10026.035} C_VEL
LIN {X 0,Y 423.146,Z 276.431,A -85,B 0,C 180,E1 -10026.721,E2 -10026.721} C_VEL
LIN {X 0,Y 423.575,Z 263.743,A -85,B 0,C 180,E1 -10027.179,E2 -10027.179} C_VEL
LIN {X 0,Y 423.838,Z 247.885,A -85,B 0,C 180,E1 -10027.512,E2 -10027.512} C_VEL
LIN {X 0,Y 424.89,Z 171.687,A -85,B 0,C 180,E1 -10028.834,E2 -10028.834} C_VEL
LIN {X 0,Y 420.911,Z 154.51,A -85,B 0,C 180,E1 -10029.365,E2 -10029.365} C_VEL
LIN {X 0,Y 420.457,Z 152.827,A -85,B 0,C 180,E1 -10029.433,E2 -10029.433} C_VEL
LIN {X 0,Y 418.734,Z 143.594,A -85,B 0,C 180,E1 -10031.677,E2 -10031.677} C_VEL
LIN {X 0,Y 418.228,Z 141.39,A -85,B 0,C 180,E1 -10032.235,E2 -10032.235} C_VEL
LIN {X 0,Y 418.235,Z 141.39,A -85,B 0,C 180,E1 -10035.109,E2 -10035.109} C_VEL
LIN {X 0,Y 418.219,Z 141.392,A -85,B 0,C 180,E1 -10037.764,E2 -10037.764} C_VEL
LIN {X 0,Y 418.238,Z 141.389,A -85,B 0,C 180,E1 -10041.557,E2 -10041.557} C_VEL
LIN {X 0,Y 418.251,Z 141.389,A -85,B 0,C 180,E1 -10045.158,E2 -10045.158} C_VEL
LIN {X 0,Y 418.239,Z 141.388,A -85,B 0,C 180,E1 -10047.472,E2 -10047.472} C_VEL
LIN {X 0,Y 418.259,Z 141.386,A -85,B 0,C 180,E1 -10050.898,E2 -10050.898} C_VEL
LIN {X 0,Y 418.211,Z 141.391,A -85,B 0,C 180,E1 -10054.092,E2 -10054.092} C_VEL
LIN {X 0,Y 418.224,Z 141.383,A -85,B 0,C 180,E1 -10057.263,E2 -10057.263} C_VEL
LIN {X 0,Y 418.246,Z 141.386,A -85,B 0,C 180,E1 -10060.363,E2 -10060.363} C_VEL
LIN {X 0,Y 418.28,Z 141.38,A -85,B 0,C 180,E1 -10063.403,E2 -10063.403} C_VEL
LIN {X 0,Y 418.346,Z 141.371,A -85,B 0,C 180,E1 -10067.385,E2 -10067.385} C_VEL
LIN {X 0,Y 418.32,Z 141.377,A -85,B 0,C 180,E1 -10070.328,E2 -10070.328} C_VEL
LIN {X 0,Y 418.441,Z 141.354,A -85,B 0,C 180,E1 -10073.248,E2 -10073.248} C_VEL
LIN {X 0,Y 418.312,Z 141.374,A -85,B 0,C 180,E1 -10075.181,E2 -10075.181} C_VEL
LIN {X 0,Y 418.534,Z 141.344,A -85,B 0,C 180,E1 -10078.076,E2 -10078.076} C_VEL
LIN {X 0,Y 418.407,Z 141.362,A -85,B 0,C 180,E1 -10080.963,E2 -10080.963} C_VEL
LIN {X 0,Y 418.47,Z 141.347,A -85,B 0,C 180,E1 -10082.888,E2 -10082.888} C_VEL
LIN {X 0,Y 418.484,Z 141.358,A -85,B 0,C 180,E1 -10085.783,E2 -10085.783} C_VEL
LIN {X 0,Y 418.371,Z 141.364,A -85,B 0,C 180,E1 -10088.696,E2 -10088.696} C_VEL
LIN {X 0,Y 418.315,Z 141.375,A -85,B 0,C 180,E1 -10091.631,E2 -10091.631} C_VEL
LIN {X 0,Y 418.299,Z 141.376,A -85,B 0,C 180,E1 -10094.597,E2 -10094.597} C_VEL
LIN {X 0,Y 418.279,Z 141.376,A -85,B 0,C 180,E1 -10097.604,E2 -10097.604} C_VEL
LIN {X 0,Y 418.252,Z 141.383,A -85,B 0,C 180,E1 -10100.663,E2 -10100.663} C_VEL
LIN {X 0,Y 418.286,Z 141.379,A -85,B 0,C 180,E1 -10103.781,E2 -10103.781} C_VEL
LIN {X 0,Y 418.224,Z 141.385,A -85,B 0,C 180,E1 -10107.047,E2 -10107.047} C_VEL
LIN {X 0,Y 418.243,Z 141.382,A -85,B 0,C 180,E1 -10110.272,E2 -10110.272} C_VEL
LIN {X 0,Y 418.25,Z 141.38,A -85,B 0,C 180,E1 -10113.677,E2 -10113.677} C_VEL
LIN {X 0,Y 418.241,Z 141.383,A -85,B 0,C 180,E1 -10117.224,E2 -10117.224} C_VEL
LIN {X 0,Y 418.215,Z 141.392,A -85,B 0,C 180,E1 -10120.868,E2 -10120.868} C_VEL
LIN {X 0,Y 418.21,Z 141.389,A -85,B 0,C 180,E1 -10123.729,E2 -10123.729} C_VEL
LIN {X 0,Y 418.21,Z 141.395,A -85,B 0,C 180,E1 -10126.449,E2 -10126.449} C_VEL
LIN {X 0,Y 418.223,Z 141.39,A -85,B 0,C 180,E1 -10129.131,E2 -10129.131} C_VEL
LIN {X 0,Y 418.226,Z 141.385,A -85,B 0,C 180,E1 -10132.167,E2 -10132.167} C_VEL
LIN {X 0,Y 418.268,Z 141.379,A -85,B 0,C 180,E1 -10135.42,E2 -10135.42} C_VEL
LIN {X 0,Y 418.215,Z 141.394,A -85,B 0,C 180,E1 -10138.604,E2 -10138.604} C_VEL
LIN {X 0,Y 418.314,Z 141.397,A -85,B 0,C 180,E1 -10141.391,E2 -10141.391} C_VEL
LIN {X 0,Y 420.918,Z 153.362,A -85,B 0,C 180,E1 -10144.005,E2 -10144.005} C_VEL
LIN {X 0,Y 421.747,Z 158.678,A -85,B 0,C 180,E1 -10145.117,E2 -10145.117} C_VEL
LIN {X 0,Y 420.547,Z 175.994,A -85,B 0,C 180,E1 -10148.429,E2 -10148.429} C_VEL
LIN {X 0,Y 419.89,Z 187.575,A -85,B 0,C 180,E1 -10150.594,E2 -10150.594} C_VEL
LIN {X 0,Y 423.873,Z 211.756,A -85,B 0,C 180,E1 -10151.245,E2 -10151.245} C_VEL
LIN {X 0,Y 424.286,Z 218.064,A -85,B 0,C 180,E1 -10151.38,E2 -10151.38} C_VEL
LIN {X 0,Y 423.349,Z 296.447,A -85,B 0,C 180,E1 -10152.769,E2 -10152.769} C_VEL
LIN {X 0,Y 422.752,Z 309.554,A -85,B 0,C 180,E1 -10153.18,E2 -10153.18} C_VEL
LIN {X 0,Y 422.002,Z 322.756,A -85,B 0,C 180,E1 -10153.802,E2 -10153.802} C_VEL
LIN {X 0,Y 421.259,Z 333.884,A -85,B 0,C 180,E1 -10154.518,E2 -10154.518} C_VEL
LIN {X 0,Y 420.395,Z 345.469,A -85,B 0,C 180,E1 -10155.477,E2 -10155.477} C_VEL
LIN {X 0,Y 419.568,Z 355.92,A -85,B 0,C 180,E1 -10156.561,E2 -10156.561} C_VEL
LIN {X 0,Y 418.97,Z 364.486,A -85,B 0,C 180,E1 -10157.65,E2 -10157.65} C_VEL
LIN {X 0,Y 418.306,Z 372.405,A -85,B 0,C 180,E1 -10158.859,E2 -10158.859} C_VEL
LIN {X 0,Y 417.761,Z 380.183,A -85,B 0,C 180,E1 -10160.315,E2 -10160.315} C_VEL
LIN {X 0,Y 417.431,Z 386.441,A -85,B 0,C 180,E1 -10161.772,E2 -10161.772} C_VEL
LIN {X 0,Y 417.177,Z 391.427,A -85,B 0,C 180,E1 -10163.227,E2 -10163.227} C_VEL
LIN {X 0,Y 417.088,Z 395.29,A -85,B 0,C 180,E1 -10164.682,E2 -10164.682} C_VEL
LIN {X 0,Y 417.022,Z 398.126,A -85,B 0,C 180,E1 -10166.135,E2 -10166.135} C_VEL
LIN {X 0,Y 417.074,Z 399.476,A -85,B 0,C 180,E1 -10167.102,E2 -10167.102} C_VEL
LIN {X 0,Y 417.092,Z 400.429,A -85,B 0,C 180,E1 -10168.069,E2 -10168.069} C_VEL
LIN {X 0,Y 417.06,Z 400.98,A -85,B 0,C 180,E1 -10169.034,E2 -10169.034} C_VEL
LIN {X 0,Y 417.059,Z 401.095,A -85,B 0,C 180,E1 -10170,E2 -10170} C_VEL
LIN {X 0,Y 417.093,Z 400.152,A -85,B 0,C 180,E1 -10171.931,E2 -10171.931} C_VEL
LIN {X 0,Y 417.092,Z 399.084,A -85,B 0,C 180,E1 -10172.897,E2 -10172.897} C_VEL
LIN {X 0,Y 417.026,Z 397.553,A -85,B 0,C 180,E1 -10173.865,E2 -10173.865} C_VEL
LIN {X 0,Y 417.104,Z 394.468,A -85,B 0,C 180,E1 -10175.317,E2 -10175.317} C_VEL
LIN {X 0,Y 417.159,Z 390.304,A -85,B 0,C 180,E1 -10176.773,E2 -10176.773} C_VEL
